	        //Funkcja cykliczna
	        IF NOT #State.inputFlag AND NOT #State.outputFlag THEN
	            IF #Reset THEN
	                #Status.Error := FALSE;
	                #Status.ErrorStatus := 16#0000;
	                IF NOT #Valve.Sensors.In THEN
	                    "changeState"(newState := #S_GO_IN,
	                                  Data := #State);
	                ELSE
	                    "changeState"(newState := #S_IDLE,
	                                  Data := #State);
	                END_IF;
	            END_IF;
	        END_IF;
	        
	        //Funkcja wyjściowa 
	        IF #State.outputFlag THEN
	            ;
	        END_IF;
	        
	    #S_GO_IN:
	        //Funkcja wejścia
	        IF #State.inputFlag AND NOT #State.outputFlag THEN
	            #State.name := 'CHOWANIE SILOWNIKA';
	            #Status.Busy := TRUE;
	            #Status.Ready := FALSE;
	           // #Status.Done := FALSE;
	            #Status.Error := FALSE;
	            #Valve.Coils.In := TRUE;
	            #Valve.Coils.Out := FALSE;
	            RESET_TIMER(#Timers.GoOut.Timer);
	            
	            #Timers.SetIn.IN := TRUE;
	            #Timers.GoOut.IN := TRUE;
	        END_IF;
	        
	        //Funkcja cykliczna
	        IF NOT #State.inputFlag AND NOT #State.outputFlag THEN
	            IF #Valve.Sensors.In AND (NOT #FirstTry OR NOT #SecondPush ) THEN
	                #Execute := FALSE;
	                "changeState"(newState := #S_IDLE,
	                              Data := #State);
	            END_IF;
	            
	            IF #SecondPush AND #FirstTry AND #Timers.GoOut.Timer.Q THEN
	                #FirstTry := FALSE;
	                "changeState"(newState := #S_GO_OUT,
	                              Data := #State);
	            END_IF;
	            
	            
	            
	            IF #Timers.SetIn.Timer.Q THEN
	                #Status.ErrorStatus := #WatchdogIn;
	                "changeState"(newState := #S_ERROR,
	                              Data := #State);
	            END_IF;
	        END_IF;
	        
	        //Funkcja wyjściowa 
	        IF #State.outputFlag THEN
	            #Valve.Coils.In := FALSE;
	            #Timers.SetIn.IN := FALSE;
	            #Timers.GoOut.IN := FALSE;
	        END_IF;
	        
	    #S_GO_OUT:
	        //Funkcja wejścia
	        IF #State.inputFlag AND NOT #State.outputFlag THEN
	            #State.name := 'WYSUNIECIE SILOWNIKA';
	            #Status.Busy := TRUE;
	            #Status.Ready := FALSE;
	            #Status.Done := FALSE;
	            #Status.Error := FALSE;
	            #Valve.Coils.In := FALSE;
	            #Valve.Coils.Out := TRUE;
	            RESET_TIMER(#Timers.Stamping.Timer);
	            RESET_TIMER(#Timers.SetOut.Timer);
	            RESET_TIMER(#Timers.Stamping.Timer);
	            #Timers.SetOut.IN := TRUE;
	        END_IF;
	        
	        //Funkcja cykliczna
	        IF NOT #State.inputFlag AND NOT #State.outputFlag THEN
	            
	            IF #Timers.Stamping.Timer.Q AND #FirstTry THEN
	                #Execute := FALSE;
	                "changeState"(newState := #S_GO_IN,
	                              Data := #State);
	            END_IF;
	            
	            IF #Timers.SecondPush.Timer.Q AND NOT #FirstTry THEN
	                #Execute := FALSE;
	                "changeState"(newState := #S_GO_IN,
	                              Data := #State);
	            END_IF;
	            
	            IF #Timers.SetOut.Timer.Q THEN
	                #Status.ErrorStatus := #WatchdogOut;
	                "changeState"(newState := #S_ERROR,
	                              Data := #State);
	            END_IF;
	        END_IF;
	        
	        //Funkcja wyjściowa 
	        IF #State.outputFlag THEN
	            RESET_TIMER(#Timers.Stamping.Timer);
	            RESET_TIMER(#Timers.SetOut.Timer);
	            RESET_TIMER(#Timers.SecondPush.Timer);
	            #Valve.Coils.Out := FALSE;
	            #Timers.SetOut.IN := FALSE;
	        END_IF;
	END_CASE;
	
	IF (#Timers.SetOut.Timer.ET > #TimerMax AND #FirstTry) THEN
	    #ITV.Sensor.Analog.SetValue := #MaxPreasure;
	ELSIF (#Timers.SetOut.Timer.ET > #TimerSecondPush AND NOT #FirstTry) THEN
	    #ITV.Sensor.Analog.SetValue := #PreasureSecondPush;
	ELSIF #Valve.Coils.In THEN
	    #ITV.Sensor.Analog.SetValue := 3.0;
	ELSE
	    #ITV.Sensor.Analog.SetValue := #RegularPreasure;
	END_IF;
	
	REGION Change state
	    IF #State.inputFlag AND NOT #State.outputFlag THEN
	        #State.inputFlag := FALSE;
	    END_IF;
	    #State.outputFlag := FALSE;
	END_REGION
END_FUNCTION_BLOCK

FUNCTION "changeState" : Void
{ S7_Optimized_Access := 'TRUE' }
VERSION : 0.1
   VAR_INPUT 
      newState : Int;
   END_VAR

   VAR_IN_OUT 
      Data : "s_changeState";
   END_VAR


BEGIN
	IF #Data.state <> #newState THEN
	    #Data.oldState := #Data.state;
	    #Data.state := #newState;
	    #Data.inputFlag := TRUE;
	    #Data.outputFlag := TRUE;
	END_IF;
	
END_FUNCTION

FUNCTION "FC_004_ModularConvoyers" : Void   // FC11, LAD
{ S7_Optimized_Access := 'TRUE' }
// stored: SetENOAutomatically false
BEGIN

REGION Network 1 (SCL)
   //************************************************************
   //===Author: Mateusz Połojko
   //-----Linkedin: https://pl.linkedin.com/in/mateusz-po%C5%82ojko-52a3541b1
   //-----Github: https://github.com/Bhazel95
   //===Description:
   //-----Control of the transporter and executive modules
   //===Customer:
   //-----Apator Powogaz S.A.
   //************************************************************
END_REGION

REGION Network 2
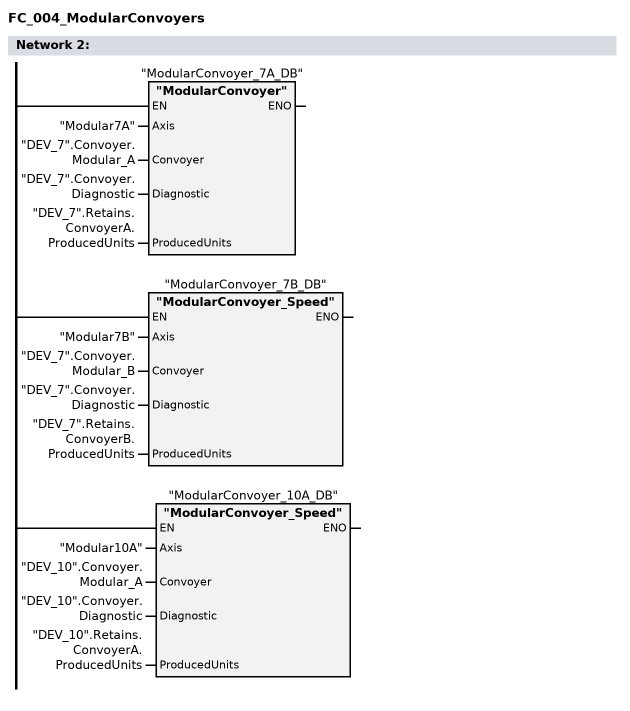
   RUNG wire#powerrail
      "ModularConvoyer_7A_DB"(Axis := "Modular7A", Convoyer := "DEV_7".Convoyer.Modular_A, Diagnostic := "DEV_7".Convoyer.Diagnostic, ProducedUnits := "DEV_7".Retains.ConvoyerA.ProducedUnits)
   END_RUNG
   RUNG wire#powerrail
      "ModularConvoyer_7B_DB"(Axis := "Modular7B", Convoyer := "DEV_7".Convoyer.Modular_B, Diagnostic := "DEV_7".Convoyer.Diagnostic, ProducedUnits := "DEV_7".Retains.ConvoyerB.ProducedUnits)
   END_RUNG
   RUNG wire#powerrail
      "ModularConvoyer_10A_DB"(Axis := "Modular10A", Convoyer := "DEV_10".Convoyer.Modular_A, Diagnostic := "DEV_10".Convoyer.Diagnostic, ProducedUnits := "DEV_10".Retains.ConvoyerA.ProducedUnits)
   END_RUNG
   // the same network as SCL:
   "ModularConvoyer_7A_DB"(Axis := "Modular7A",   // "ModularConvoyer"
                           Convoyer := "DEV_7".Convoyer.Modular_A,
                           Diagnostic := "DEV_7".Convoyer.Diagnostic,
                           ProducedUnits := "DEV_7".Retains.ConvoyerA.ProducedUnits);
   "ModularConvoyer_7B_DB"(Axis := "Modular7B",   // "ModularConvoyer_Speed"
                           Convoyer := "DEV_7".Convoyer.Modular_B,
                           Diagnostic := "DEV_7".Convoyer.Diagnostic,
                           ProducedUnits := "DEV_7".Retains.ConvoyerB.ProducedUnits);
   "ModularConvoyer_10A_DB"(Axis := "Modular10A",   // "ModularConvoyer_Speed"
                           Convoyer := "DEV_10".Convoyer.Modular_A,
                           Diagnostic := "DEV_10".Convoyer.Diagnostic,
                           ProducedUnits := "DEV_10".Retains.ConvoyerA.ProducedUnits);
END_REGION
END_FUNCTION

FUNCTION_BLOCK "ModularConvoyer"
{ S7_Optimized_Access := 'TRUE' }
VERSION : 0.1
   VAR_INPUT 
      Axis {InstructionName := 'TO_PositioningAxis'; LibVersion := '7.0'} : TO_PositioningAxis;
   END_VAR

   VAR_IN_OUT 
      Convoyer : "Modular_10";
      Diagnostic : "DiagnosticMainCabinet";
      ProducedUnits : DInt;
   END_VAR

   VAR 
      R_TRIG_CriticalError {InstructionName := 'R_TRIG'; LibVersion := '1.0'; ExternalAccessible := 'False'; ExternalVisible := 'False'; ExternalWritable := 'False'; S7_SetPoint := 'False'} : R_TRIG;
      R_TRIG_StampingDone {InstructionName := 'R_TRIG'; LibVersion := '1.0'; ExternalAccessible := 'False'; ExternalVisible := 'False'; ExternalWritable := 'False'; S7_SetPoint := 'False'} : R_TRIG;
      R_TRIG_CameraDone {InstructionName := 'R_TRIG'; LibVersion := '1.0'; ExternalAccessible := 'False'; ExternalVisible := 'False'; ExternalWritable := 'False'; S7_SetPoint := 'False'} : R_TRIG;
      R_TRIG_SortingDone {InstructionName := 'R_TRIG'; LibVersion := '1.0'; ExternalAccessible := 'False'; ExternalVisible := 'False'; ExternalWritable := 'False'; S7_SetPoint := 'False'} : R_TRIG;
      R_TRIG_ConvoyerDone {InstructionName := 'R_TRIG'; LibVersion := '1.0'; ExternalAccessible := 'False'; ExternalVisible := 'False'; ExternalWritable := 'False'; S7_SetPoint := 'False'} : R_TRIG;
      R_TRIG_Stop {InstructionName := 'R_TRIG'; LibVersion := '1.0'; ExternalAccessible := 'False'; ExternalVisible := 'False'; ExternalWritable := 'False'; S7_SetPoint := 'False'} : R_TRIG;
      State { S7_SetPoint := 'False'} : "s_changeState";
      Local : Struct
         AutoMode : Bool;
         Buttons : Struct
            START : Bool;
            RESET : Bool;
            STOP : Bool;
         END_STRUCT;
         PermissionToStart : Bool;
         PermissionGoBack : Bool;
         ActionDone : Struct
            Stamping : Bool;
            Camera : Bool;
            Sorting : Bool;
         END_STRUCT;
         Execute : Struct
            Stamping : Bool;
            Camera : Bool;
            Sorting : Bool;
            Convoyer : Bool;
            Blow : Bool;
         END_STRUCT;
         ActionToDo : Struct
            Stamping : Bool;
            Camera : Bool;
            Blow : Bool;
            PreCamera : Array[0..1] of Bool;
         END_STRUCT;
         DoubleStampingDone : Bool;
         StampingTime : Time;
         isMoved : Bool;
         backwardProcess : Bool;
      END_STRUCT;
      Timers : Struct
         WatchdogGoModules { S7_SetPoint := 'False'} : "s_TON";
         WatchdogGoConvoyer : "s_TON";
         Delay : "s_TON";
         DoubleStamp : "s_TON";
         UnloadTimer {InstructionName := 'TON_TIME'; LibVersion := '1.0'; ExternalAccessible := 'False'; ExternalVisible := 'False'; ExternalWritable := 'False'; S7_SetPoint := 'False'} : TON_TIME;
         OskarDelay : "s_TON";
         GoBackwardEnable : "s_TON";
         GoBackward : "s_TON";
      END_STRUCT;
      CameraConnectionTCP_Instance { ExternalAccessible := 'False'; ExternalVisible := 'False'; ExternalWritable := 'False'; S7_SetPoint := 'False'} : "CameraConnectionTCP";
      PositioningAxis_Instance { ExternalAccessible := 'False'; ExternalVisible := 'False'; ExternalWritable := 'False'; S7_SetPoint := 'False'} : "ModularAxis";
      Blow_Instance : "Blow";
      Stamping_Instance : "Stamping";
   END_VAR

   VAR CONSTANT 
      S_IDLE : Int := 0;
      S_ERROR : Int := 20;
      S_GO_CONVOYER : Int := 30;
      S_GO_MODULES : Int := 40;
      S_GO_BACK : Int := 50;
      TEST : Int := 100;
      E_MODULES_TIMEOUT : Word := 16#8000;
      E_CONVOYER_TIMEOUT : Word := 16#8001;
   END_VAR


BEGIN
	//************************************************************
	//===Author: Mateusz Połojko
	//-----Linkedin: https://pl.linkedin.com/in/mateusz-po%C5%82ojko-52a3541b1
	//-----Github: https://github.com/Bhazel95
	//===Description:
	//-----Main function block for convoyer + executive modules control
	//===Customer:
	//-----Apator Powogaz S.A.
	//************************************************************
	
	REGION R/F_TRIG
	    #R_TRIG_CriticalError(CLK := NOT #Convoyer.Safety.SafetyOK OR #PositioningAxis_Instance.Status.Error);
	    #R_TRIG_StampingDone(CLK := #Stamping_Instance.Status.Done);
	    #R_TRIG_CameraDone(CLK := #CameraConnectionTCP_Instance.Status.Done);
	    #R_TRIG_SortingDone(CLK := #Convoyer.SortingStatus.Done);
	    #R_TRIG_ConvoyerDone(CLK := #PositioningAxis_Instance.Status.Ready);
	    #R_TRIG_Stop(CLK := #Local.Buttons.STOP AND #Local.AutoMode);
	END_REGION
	
	REGION Timers
	    //WATCHDOG MACHINE START
	    #Timers.WatchdogGoModules.PT := T#15S;
	    #Timers.WatchdogGoModules.Timer(IN := #Timers.WatchdogGoModules.IN,
	                                    PT := #Timers.WatchdogGoModules.PT);
	    #Timers.WatchdogGoConvoyer.PT := T#10S;
	    #Timers.WatchdogGoConvoyer.Timer(IN := #Timers.WatchdogGoConvoyer.IN,
	                                     PT := #Timers.WatchdogGoConvoyer.PT);
	    #Timers.Delay.PT := T#7S;
	    #Timers.Delay.Timer(IN := #Timers.Delay.IN,
	                        PT := #Timers.Delay.PT);
	    
	    #Timers.DoubleStamp.PT := T#500MS;
	    #Timers.DoubleStamp.Timer(IN := #Timers.DoubleStamp.IN,
	                              PT := #Timers.DoubleStamp.PT);
	    
	    #Timers.OskarDelay.PT := T#5000MS;
	    #Timers.OskarDelay.Timer(IN := #Timers.OskarDelay.IN,
	                             PT := #Timers.OskarDelay.PT);
	    
	    #Timers.GoBackwardEnable.PT := T#3000MS;
	    #Timers.GoBackwardEnable.Timer(IN := #Convoyer.ButtonControl.ButtonBoxLeft.ButtonReset OR #Convoyer.ButtonControl.ButtonBoxRight.ButtonReset,
	                                   PT := #Timers.GoBackwardEnable.PT);
	    
	    #Timers.GoBackward.PT := T#2000MS;
	    #Timers.GoBackward.Timer(IN := #Timers.GoBackward.IN,
	                             PT := #Timers.GoBackward.PT);
	    
	    #Timers.UnloadTimer(IN := NOT #Convoyer.Sensors.UnloadingPresence,
	                        PT := T#1000MS);
	END_REGION
	
	//Permission to start
	#Local.PermissionToStart := #Diagnostic.DiagnosticOK AND NOT #Convoyer.Alarms.Fault24V AND #Convoyer.Safety.SafetyOK
	AND NOT #Convoyer.Alarms.Present AND #Convoyer.Pneumatics.Stamping.Sensors.In AND #Convoyer.Safety.LightCurtain_Stamping
	AND NOT #Convoyer.Pneumatics.Stamping.Sensors.Out AND (#Convoyer.CameraStatus.Ready OR NOT #Convoyer.HMI.Camera.Enable)
	AND #Convoyer.MotorStatus.Ready AND #Convoyer.Sensors.Stamp_Check_1 AND #Convoyer.Sensors.UnloadingPresence AND #Convoyer.Sensors.Span;
	
	#Local.PermissionGoBack := #Diagnostic.DiagnosticOK AND #Convoyer.Safety.SafetyOK
	AND NOT #Convoyer.Alarms.Present AND #Convoyer.Pneumatics.Stamping.Sensors.In
	AND NOT #Convoyer.Pneumatics.Stamping.Sensors.Out AND #Convoyer.MotorStatus.Ready AND #Convoyer.Sensors.Stamp_Check_1 AND #Convoyer.Sensors.UnloadingPresence AND #Convoyer.Sensors.Span AND #Convoyer.Sensors.JogBack;
	
	//Start button
	#Local.Buttons.START := #Convoyer.ButtonControl.ButtonBoxLeft.ButtonStart OR #Convoyer.ButtonControl.ButtonBoxRight.ButtonStart OR #Convoyer.HMI.Buttons.Start;
	//Stop button
	#Local.Buttons.STOP := #Convoyer.ButtonControl.ButtonBoxLeft.ButtonStop OR #Convoyer.ButtonControl.ButtonBoxRight.ButtonStop OR #Convoyer.HMI.Buttons.Stop;
	//Reset button
	#Local.Buttons.RESET := #Convoyer.ButtonControl.ButtonBoxLeft.ButtonReset OR #Convoyer.ButtonControl.ButtonBoxRight.ButtonReset OR #Convoyer.ButtonControl.CabinetBox.ButtonReset;
	
	CASE #State.state OF
	    #S_IDLE:
	        //Funkcja wejścia
	        IF #State.inputFlag AND NOT #State.outputFlag THEN
	            #Convoyer.ConvoyerStatus.Busy := FALSE;
	            #Convoyer.ConvoyerStatus.Done := FALSE;
	            #Convoyer.ConvoyerStatus.Error := FALSE;
	            #Convoyer.ConvoyerStatus.ErrorStatus := 16#0000;
	            #Convoyer.ConvoyerStatus.Ready := TRUE;
	        END_IF;
	        
	        //Funkcja cykliczna
	        IF NOT #State.inputFlag AND NOT #State.outputFlag THEN
	            //ZABEZPIECZENIE PRZED MANUALNYM RUSZENIEM TRANSPORTERA
	            IF #Convoyer.MotorControl.MC_MOVEJOG.JogBackward OR #Convoyer.MotorControl.MC_MOVEJOG.JogForward THEN
	                #Local.isMoved := TRUE;
	            END_IF;
	            IF #Convoyer.Safety.LightCurtain_Stamping AND #Local.PermissionToStart AND (#Local.Buttons.START OR #Local.AutoMode) AND NOT #Local.Buttons.STOP AND NOT #Local.Buttons.RESET THEN
	                #Local.AutoMode := TRUE;
	                IF ((NOT #Convoyer.Sensors.StampingPresence AND NOT #Local.ActionDone.Stamping) OR (NOT #Convoyer.Sensors.CameraPresence AND NOT #Local.ActionDone.Camera)) AND NOT #Local.isMoved THEN
	                    "changeState"(newState := #S_GO_MODULES,
	                                  Data := #State);
	                ELSIF ((#Local.ActionDone.Stamping OR #Convoyer.Sensors.StampingPresence) AND (#Local.ActionDone.Camera OR #Convoyer.Sensors.CameraPresence)) OR #Local.isMoved THEN
	                    "changeState"(newState := #S_GO_CONVOYER,
	                                  Data := #State);
	                END_IF;
	            END_IF;
	            //COFANIE TRANSPORTERA
	            IF NOT #Local.AutoMode AND #Local.PermissionGoBack AND #Timers.GoBackwardEnable.Timer.Q AND NOT #Local.Buttons.START AND NOT #Local.Buttons.STOP THEN
	                #Local.isMoved := TRUE;
	                "changeState"(newState := #S_GO_BACK,
	                              Data := #State);
	            END_IF;
	            
	        END_IF;
	        
	        //Funkcja wyjściowa 
	        IF #State.outputFlag THEN
	            #Convoyer.ConvoyerStatus.Ready := FALSE;
	            #Convoyer.ConvoyerStatus.Busy := TRUE;
	        END_IF;
	        
	    #S_ERROR:
	        //Funkcja wejścia
	        IF #State.inputFlag AND NOT #State.outputFlag THEN
	            #Convoyer.ConvoyerStatus.Busy := FALSE;
	            #Convoyer.ConvoyerStatus.Done := FALSE;
	            #Convoyer.ConvoyerStatus.Error := TRUE;
	            #Convoyer.ConvoyerStatus.Ready := FALSE;
	            #Timers.WatchdogGoConvoyer.IN := FALSE;
	            #Timers.WatchdogGoModules.IN := FALSE;
	            #Local.Execute.Convoyer := FALSE;
	            #Local.Execute.Stamping := FALSE;
	            #Local.Execute.Camera := FALSE;
	            //#Local.ActionDone.Camera := FALSE;
	            #Local.AutoMode := FALSE;
	        END_IF;
	        
	        //Funkcja cykliczna
	        IF NOT #State.inputFlag AND NOT #State.outputFlag THEN
	            IF #Local.Buttons.RESET AND NOT #Convoyer.Alarms.Present AND #Convoyer.Safety.SafetyOK
	                AND (#CameraConnectionTCP_Instance.Status.Ready OR NOT #Convoyer.HMI.Camera.Enable) AND #PositioningAxis_Instance.Status.Ready
	                AND (#Stamping_Instance.Status.Ready OR NOT #Convoyer.HMI.Stamping.Enable) AND #Local.PermissionToStart THEN
	                #Convoyer.ConvoyerStatus.Error := FALSE;
	                "changeState"(newState := #S_IDLE,
	                              Data := #State);
	            END_IF;
	        END_IF;
	        
	        //Funkcja wyjściowa 
	        IF #State.outputFlag THEN
	            ;
	        END_IF;
	        
	    #S_GO_CONVOYER:
	        //Funkcja wejścia
	        IF #State.inputFlag AND NOT #State.outputFlag THEN
	            #Timers.WatchdogGoConvoyer.IN := TRUE;
	            #Local.ActionDone.Stamping := FALSE;
	            #Local.ActionDone.Camera := FALSE;
	            #Local.ActionDone.Sorting := FALSE;
	            #Local.ActionToDo.PreCamera[1] := #Local.ActionToDo.PreCamera[0];
	            #Local.Execute.Convoyer := TRUE;
	        END_IF;
	        
	        //Funkcja cykliczna
	        IF NOT #State.inputFlag AND NOT #State.outputFlag THEN
	            IF #R_TRIG_ConvoyerDone.Q THEN
	                #Local.isMoved := FALSE;
	                IF NOT #Local.AutoMode OR NOT #Convoyer.Safety.LightCurtain_Stamping THEN
	                    "changeState"(newState := #S_IDLE,
	                                  Data := #State);
	                ELSE
	                    "changeState"(newState := #S_GO_MODULES,
	                                  Data := #State);
	                END_IF;
	            END_IF;
	            IF #PositioningAxis_Instance.Status.Error THEN
	                "changeState"(newState := #S_ERROR,
	                              Data := #State);
	            END_IF;
	            //WATCHDOG
	            IF #Timers.WatchdogGoConvoyer.Timer.Q THEN
	                #PositioningAxis_Instance.Status.ErrorStatus := #E_CONVOYER_TIMEOUT;
	                "changeState"(newState := #S_ERROR,
	                              Data := #State);
	            END_IF;
	        END_IF;
	        
	        //Funkcja wyjściowa 
	        IF #State.outputFlag THEN
	            #Local.Execute.Convoyer := FALSE;
	            #Local.ActionDone.Stamping := FALSE;
	            #Local.ActionDone.Camera := FALSE;
	            #Local.ActionDone.Sorting := FALSE;
	            #Timers.WatchdogGoConvoyer.IN := FALSE;
	            #Local.Execute.Convoyer := FALSE;
	        END_IF;
	        
	    #S_GO_MODULES:
	        //Funkcja wejścia
	        IF #State.inputFlag AND NOT #State.outputFlag THEN
	            #Timers.OskarDelay.IN := TRUE;
	            #Timers.WatchdogGoModules.IN := TRUE;
	            #Timers.Delay.IN := TRUE;
	            #Local.DoubleStampingDone := FALSE;
	            IF #Convoyer.HMI.Stamping.Double THEN
	                #Local.StampingTime := T#1MS;
	            ELSE
	                #Local.StampingTime := #Convoyer.HMI.Stamping.TimerStamping;
	            END_IF;
	            #Local.Execute.Blow := #Convoyer.Sensors.BlowPresence AND #Convoyer.HMI.Blow.Enable;
	            #Local.Execute.Stamping := NOT #Local.ActionDone.Stamping AND NOT #Convoyer.Sensors.StampingPresence AND #Convoyer.HMI.Stamping.Enable;
	            
	            //TUTAJ NA DOLE
	            #Local.Execute.Camera := ((NOT #Local.ActionDone.Camera AND NOT #Convoyer.Sensors.CameraPresence) OR (#Local.ActionToDo.PreCamera[1] AND NOT #Local.ActionDone.Camera)) AND #Convoyer.HMI.Camera.Enable;
	            #Local.ActionToDo.Stamping := #Local.Execute.Stamping;
	            #Local.ActionToDo.Camera := #Local.Execute.Camera;
	            #Local.ActionToDo.PreCamera[0] := #Convoyer.Sensors.BlowPresence; //DODANE ABY ZOBACZYC CZY WYELIMINUJE BLAD BRAKU ZDJEC
	        END_IF;
	        //Funkcja cykliczna
	        IF NOT #State.inputFlag AND NOT #State.outputFlag THEN
	            REGION double stamping
	                IF #Convoyer.HMI.Stamping.Double AND NOT #Local.DoubleStampingDone AND #Timers.DoubleStamp.Timer.Q THEN
	                    #Local.StampingTime := #Convoyer.HMI.Stamping.TimerStamping;
	                    #Local.DoubleStampingDone := TRUE;
	                    #Local.Execute.Stamping := TRUE;
	                END_IF;
	            END_REGION
	            
	            IF #R_TRIG_CameraDone.Q THEN
	                #Local.ActionDone.Camera := TRUE;
	                #Local.ActionToDo.Camera := FALSE;
	                #Local.Execute.Camera := FALSE;
	            END_IF;
	            IF #R_TRIG_SortingDone.Q THEN
	                #Local.ActionDone.Sorting := TRUE;
	            END_IF;
	            IF #R_TRIG_StampingDone.Q THEN
	                #ProducedUnits := #ProducedUnits + 1;
	                IF NOT #Convoyer.HMI.Stamping.Double THEN
	                    #Local.ActionDone.Stamping := TRUE;
	                    #Local.ActionToDo.Stamping := FALSE;
	                    #Local.Execute.Stamping := FALSE;
	                ELSIF #Convoyer.HMI.Stamping.Double AND NOT #Local.DoubleStampingDone THEN
	                    #Timers.DoubleStamp.IN := TRUE;
	                    #Local.Execute.Stamping := FALSE;
	                ELSIF #Convoyer.HMI.Stamping.Double AND #Local.DoubleStampingDone THEN
	                    #Local.ActionDone.Stamping := TRUE;
	                    #Local.ActionToDo.Stamping := FALSE;
	                    #Local.Execute.Stamping := FALSE;
	                END_IF;
	            END_IF;
	            
	            //Oczekiwanie na potwierdzenia blokow  - komentarz -->> opoznienie zalaczenia ruchu stolu dla Oskara
	            IF (#Local.ActionDone.Stamping OR NOT #Local.ActionToDo.Stamping) AND (#Local.ActionDone.Camera OR NOT #Local.ActionToDo.Camera) AND NOT #Local.Execute.Blow (* AND #Timers.OskarDelay.Timer.Q *)THEN
	                IF NOT #Local.AutoMode THEN
	                    "changeState"(newState := #S_IDLE,
	                                  Data := #State);
	                ELSE
	                    IF #Local.PermissionToStart THEN
	                        "changeState"(newState := #S_GO_CONVOYER,
	                                      Data := #State);
	                    ELSE
	                        "changeState"(newState := #S_IDLE,
	                                      Data := #State);
	                    END_IF;
	                END_IF;
	            END_IF;
	            //Modules Error
	            IF (#CameraConnectionTCP_Instance.Status.Error OR #Stamping_Instance.Status.Error) AND #Timers.Delay.Timer.Q THEN
	                "changeState"(newState := #S_ERROR,
	                              Data := #State);
	            END_IF;
	            
	            //WATCHDOG
	            IF #Timers.WatchdogGoModules.Timer.Q THEN
	                #PositioningAxis_Instance.Status.ErrorStatus := #E_MODULES_TIMEOUT;
	                "changeState"(newState := #S_ERROR,
	                              Data := #State);
	            END_IF;
	        END_IF;
	        
	        //Funkcja wyjściowa 
	        IF #State.outputFlag THEN
	            #Timers.Delay.IN := FALSE;
	            #Timers.OskarDelay.IN := FALSE;
	            #Timers.DoubleStamp.IN := FALSE;
	            #Timers.WatchdogGoModules.IN := FALSE;
	            #Local.Execute.Stamping := FALSE;
	            #Local.Execute.Camera := FALSE;
	            #Local.Execute.Sorting := FALSE;
	        END_IF;
	        
	    #S_GO_BACK:
	        //Funkcja wejścia
	        IF #State.inputFlag AND NOT #State.outputFlag THEN
	            #Local.backwardProcess := TRUE;
	            #Timers.GoBackward.IN := TRUE;
	            #Local.isMoved := TRUE;
	            #Convoyer.MotorControl.MC_MOVEJOG.JogBackward := TRUE;
	            
	        END_IF;
	        
	        //Funkcja cykliczna
	        IF NOT #State.inputFlag AND NOT #State.outputFlag THEN
	            IF (#Timers.GoBackward.Timer.Q AND #Convoyer.Safety.LightCurtain_Stamping) OR NOT #Convoyer.Sensors.JogBack THEN
	                #Convoyer.MotorControl.MC_MOVEJOG.JogBackward := FALSE;
	                "changeState"(newState := #S_IDLE,
	                              Data := #State);
	            END_IF;
	        END_IF;
	        
	        //Funkcja wyjściowa 
	        IF #State.outputFlag THEN
	            #Local.backwardProcess := FALSE;
	            #Convoyer.MotorControl.MC_MOVEJOG.JogBackward := FALSE;
	            #Timers.GoBackward.IN := FALSE;
	        END_IF;
	        
	END_CASE;
	
	REGION FunctionBlocks
	    #Stamping_Instance(Reset := #Local.Buttons.RESET,
	                       SecondPush := #Convoyer.HMI.Stamping.SecondPush,
	                       TimerSecondPush := #Convoyer.HMI.Stamping.TimerSecond,
	                       PreasureSecondPush := #Convoyer.HMI.Stamping.SecondPreasure,
	                       TimerStamp := #Convoyer.HMI.Stamping.TimerStamping,
	                       TimerMax := #Convoyer.HMI.Stamping.TimerMaxPreasure,
	                       MaxPreasure := #Convoyer.HMI.Stamping.MaxPreasure,
	                       RegularPreasure := #Convoyer.HMI.Stamping.RegularPreasure,
	                       Status => #Convoyer.StampingStatus,
	                       Valve := #Convoyer.Pneumatics.Stamping,
	                       ITV := #Convoyer.Pneumatics.IVT,
	                       Execute := #Local.Execute.Stamping);
	    #CameraConnectionTCP_Instance(Enable := #Convoyer.HMI.Camera.Enable,
	                                  Execute := #Local.Execute.Camera,
	                                  Reset := #Local.Buttons.RESET,
	                                  ConnectionTimer := #Convoyer.HMI.Camera.TimerConnection,
	                                  Status => #Convoyer.CameraStatus,
	                                  Parameters := #Convoyer.CameraConnection);
	    #PositioningAxis_Instance(HomingSensor := #Convoyer.Sensors.Homing_I,
	                              Reset := #Local.Buttons.RESET,
	                              InverterOK := #Convoyer.Safety.InverterOK,
	                              Axis := #Axis,
	                              Status => #Convoyer.MotorStatus,
	                              Execute := #Local.Execute.Convoyer,
	                              PositioningAxis := #Convoyer.MotorControl);
	    #Blow_Instance(Timer := #Convoyer.HMI.Blow."Time",
	                   Execute := #Local.Execute.Blow,
	                   Coil := #Convoyer.Pneumatics.Valve.Coils.Out);
	END_REGION
	
	REGION Lights
	    //RESET BUTTON
	    #Convoyer.ButtonControl.ButtonBoxLeft.LightReset := #Convoyer.ConvoyerStatus.Error OR #Convoyer.CameraStatus.Error OR #Convoyer.StampingStatus.Error OR #Convoyer.MotorStatus.Error OR (NOT #Convoyer.Pneumatics.Stamping.Sensors.In AND #Convoyer.StampingStatus.Ready) OR (#Local.backwardProcess AND "Clock_1Hz");
	    #Convoyer.ButtonControl.ButtonBoxRight.LightReset := #Convoyer.ConvoyerStatus.Error OR #Convoyer.CameraStatus.Error OR #Convoyer.StampingStatus.Error OR #Convoyer.MotorStatus.Error OR (NOT #Convoyer.Pneumatics.Stamping.Sensors.In AND #Convoyer.StampingStatus.Ready) OR (#Local.backwardProcess AND "Clock_1Hz");
	    #Convoyer.ButtonControl.CabinetBox.LightReset := #Convoyer.ConvoyerStatus.Error OR #Convoyer.CameraStatus.Error OR #Convoyer.StampingStatus.Error OR #Convoyer.MotorStatus.Error OR (NOT #Convoyer.Pneumatics.Stamping.Sensors.In AND #Convoyer.StampingStatus.Ready);
	    //STOP BUTTON
	    #Convoyer.ButtonControl.ButtonBoxLeft.LightStop := #Convoyer.ConvoyerStatus.Busy AND NOT #Local.AutoMode;
	    #Convoyer.ButtonControl.ButtonBoxRight.LightStop := #Convoyer.ConvoyerStatus.Busy AND NOT #Local.AutoMode;
	    //START BUTTON
	    #Convoyer.ButtonControl.ButtonBoxLeft.LightStart := #Convoyer.ConvoyerStatus.Ready AND #Local.PermissionToStart AND NOT #Local.AutoMode;
	    #Convoyer.ButtonControl.ButtonBoxRight.LightStart := #Convoyer.ConvoyerStatus.Ready AND #Local.PermissionToStart AND NOT #Local.AutoMode;
	    //ANDON 
	    #Convoyer.Lights.Red := #Convoyer.ConvoyerStatus.Error OR #Convoyer.CameraStatus.Error OR #Convoyer.StampingStatus.Error OR #Convoyer.MotorStatus.Error;
	    #Convoyer.Lights.Green := #Convoyer.ConvoyerStatus.Busy OR #Local.AutoMode;
	    #Convoyer.Lights.Blue := #Convoyer.ConvoyerStatus.Ready AND #Local.PermissionToStart AND NOT #Local.AutoMode;
	    #Convoyer.Lights.Orange := #Timers.UnloadTimer.Q;
	END_REGION
	
	//Set AutoMode off
	IF #R_TRIG_Stop.Q THEN
	    #Local.AutoMode := FALSE;
	END_IF;
	
	//Error trig
	IF #R_TRIG_CriticalError.Q THEN
	    IF NOT #PositioningAxis_Instance.Status.Done THEN
	        #Local.isMoved := TRUE;
	    END_IF;
	    
	    "changeState"(newState := #S_ERROR,
	                  Data := #State);
	END_IF;
	
	REGION Change state
	    IF #State.inputFlag AND NOT #State.outputFlag THEN
	        #State.inputFlag := FALSE;
	    END_IF;
	    #State.outputFlag := FALSE;
	END_REGION
END_FUNCTION_BLOCK

FUNCTION_BLOCK "CameraConnectionTCP"   // FB2, LAD
{ S7_Optimized_Access := 'TRUE' }
// stored: MemoryReserve 100, SetENOAutomatically false
   VAR_INPUT
      Enable : Bool;
      Execute : Bool;
      Reset : Bool;
      ConnectionTimer : Time;
   END_VAR
   VAR_OUTPUT
      Status : "Status";
   END_VAR
   VAR_IN_OUT
      Parameters : TCON_IP_v4;
   END_VAR
   VAR
      TCON_Instance { ExternalAccessible := 'False'; ExternalVisible := 'False'; ExternalWritable := 'False'} : TCON;
      TDISCON_Instance { ExternalAccessible := 'False'; ExternalVisible := 'False'; ExternalWritable := 'False'} : TDISCON;
      TRCV_Instance { ExternalAccessible := 'False'; ExternalVisible := 'False'; ExternalWritable := 'False'} : TRCV;
      TSEND_Instance { ExternalAccessible := 'False'; ExternalVisible := 'False'; ExternalWritable := 'False'} : TSEND;
      Connection : Struct
         TCON : Struct
            REQ : Bool;
            BUSY : Bool;
            DONE : Bool;
            ERROR : Bool;
            STATUS : Word;
            CONNECTION_DATA : Struct
               InterfaceID : HW_ANY := 64;
               ID : HW_ANY := 1;
               ConnectionType : Byte := 16#0B;
               ActiveEstablished : Bool := false;
               RemodeAddress { S7_SetPoint := 'True'} : IP_V4;
               RemotePort : UInt;
               LocalPort : UInt := 2000;
            END_STRUCT;
         END_STRUCT;
         TDISCON : Struct
            REQ : Bool;
            BUSY : Bool;
            DONE : Bool;
            ERROR : Bool;
            STATUS : Word;
         END_STRUCT;
         TSEND : Struct
            REQ : Bool;
            LEN : UDInt;
            BUSY : Bool;
            DONE : Bool;
            ERROR : Bool;
            STATUS : Word;
         END_STRUCT;
         TRVC : Struct
            ENABLE : Bool;
            ADHOC : Bool := TRUE;
            LEN : UDInt;
            NDR : Bool;
            BUSY : Bool;
            RVC_LEN : UDInt;
            ERROR : Bool;
            STATUS : Word;
         END_STRUCT;
      END_STRUCT;
      Data : Struct
         RVC : Array[0..999] of Byte;
         SEND : Array[0..999] of Byte;
      END_STRUCT;
      State : "s_changeState";
      Timers : Struct
         WatchdogInit : "s_TON";
         WatchdogCamera : "s_TON";
         WatchdogInitRVC { S7_SetPoint := 'True'} : "s_TON";
         WatchdogMachineStart { S7_SetPoint := 'True'} : "s_TON";
      END_STRUCT;
      MessageGenerating : Struct
         i : Int;
         len : DInt;
         "string" : String[100];
         chars : Array[0..99] of Char;
      END_STRUCT;
      Local : Struct
         MessageSent : Bool;
         MessageSentCounter : SInt;
         prevState : Int;
      END_STRUCT;
      F_TRIG_Enable { ExternalAccessible := 'False'; ExternalVisible := 'False'; ExternalWritable := 'False'} : F_TRIG;
      R_TRIG_Execute { ExternalAccessible := 'False'; ExternalVisible := 'False'; ExternalWritable := 'False'} : R_TRIG;
      R_TRIG_Enable { ExternalAccessible := 'False'; ExternalVisible := 'False'; ExternalWritable := 'False'} : R_TRIG;
      Connected : Bool;
      DebugCounter : DInt;
   END_VAR
   VAR CONSTANT
      S_INITIALIZE : Int := 1;
      S_DISCONNECT : Int := 10;
      S_ERROR : Int := 20;
      S_ENABLE_RVC : Int := 30;
      S_MACHINE_START : Int := 40;
      S_IDLE : Int := 50;
      S_START_CAMERA : Int := 60;
      S_REPEAT : Int := 70;
      STATE_TEST : Int := 100;
      COMAND_SEND_MACHINE_START : String := 'command: machine_start';
      COMMAND_RVC_MACHINE_START : String := 'command: camera_ready';
      COMMAND_SEND_START_CONTROL : String := 'command: start_control';
      COMMAND_RVC_CONTROL_DONE : String := 'command: control_done';
      E_CONNECTION_TIMEOUT : Word := 16#8000;
      E_WRONG_RESPONSE_MACHINE_START : Word := 16#8001;
      E_START_MACHINE_NOT_SENT : Word := 16#8002;
      E_START_MACHINE_NO_RESPONSE : Word := 16#8003;
      E_WRONG_RESPONSE_CAMERA : Word := 16#8004;
      E_CAMERA_NO_RESPONSE : Word := 16#8005;
      E_CAMERA_NOT_SENT : Word := 16#8006;
      E_TRCV_ERROR : Word := 16#8007;
      E_TRCV_TIMEOUT : Word := 16#8008;
      E_TCON_ERROR : Word := 16#8009;
      E_TDISCON_ERROR : Word := 16#8010;
      E_TSEND_ERROR : Word := 16#8011;
   END_VAR
   // Connection.TCON.CONNECTION_DATA.RemodeAddress.ADDR[1] := 192;
   // Connection.TCON.CONNECTION_DATA.RemodeAddress.ADDR[2] := 168;
   // Connection.TCON.CONNECTION_DATA.RemodeAddress.ADDR[3] := 0;
   // Connection.TCON.CONNECTION_DATA.RemodeAddress.ADDR[4] := 69;
BEGIN

REGION Network 1 (SCL)
   //************************************************************
   //===Author: Mateusz Połojko
   //-----Linkedin: https://pl.linkedin.com/in/mateusz-po%C5%82ojko-52a3541b1
   //-----Github: https://github.com/Bhazel95
   //===Description:
   //-----Camera control via TCP/IP
   //===Customer:
   //-----Apator Powogaz S.A.
   //************************************************************
END_REGION

REGION Network 2
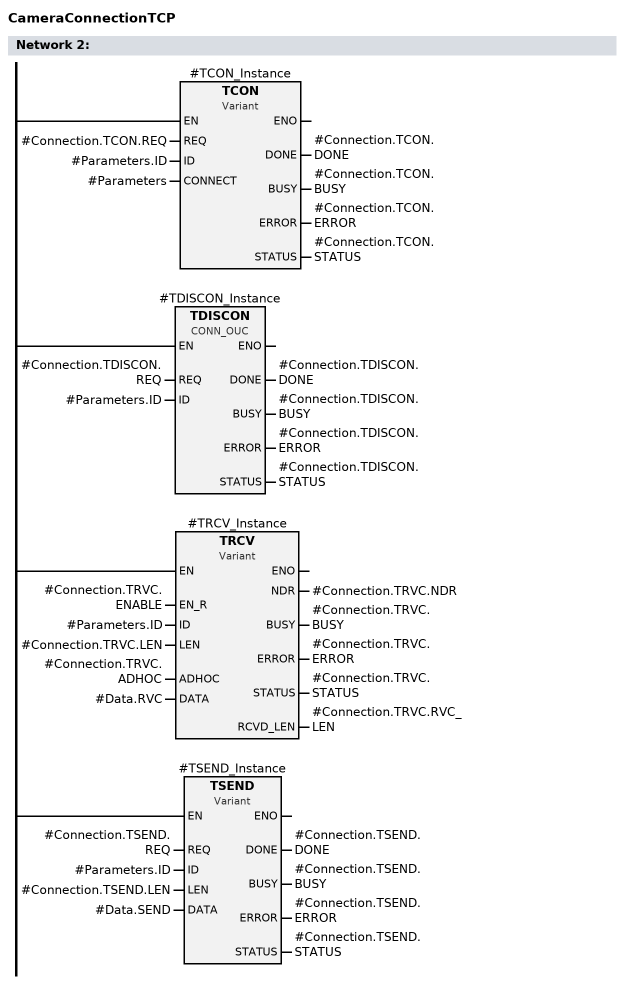
   RUNG wire#powerrail
      { S7_Templates := "[con_type := Variant, id_type := CONN_OUC]" } #TCON_Instance.TCON(REQ := #Connection.TCON.REQ, ID := #Parameters.ID, CONNECT := #Parameters, DONE => #Connection.TCON.DONE, BUSY => #Connection.TCON.BUSY, ERROR => #Connection.TCON.ERROR, STATUS => #Connection.TCON.STATUS)
   END_RUNG
   RUNG wire#powerrail
      { S7_Templates := "id_type := CONN_OUC" } #TDISCON_Instance.TDISCON(REQ := #Connection.TDISCON.REQ, ID := #Parameters.ID, DONE => #Connection.TDISCON.DONE, BUSY => #Connection.TDISCON.BUSY, ERROR => #Connection.TDISCON.ERROR, STATUS => #Connection.TDISCON.STATUS)
   END_RUNG
   RUNG wire#powerrail
      { S7_Templates := "[card := 1, ptr_type := Variant, value_type := UDInt, id_type := CONN_OUC]" } #TRCV_Instance.TRCV(EN_R := #Connection.TRVC.ENABLE, ID := #Parameters.ID, LEN := #Connection.TRVC.LEN, ADHOC := #Connection.TRVC.ADHOC, DATA := #Data.RVC, NDR => #Connection.TRVC.NDR, BUSY => #Connection.TRVC.BUSY, ERROR => #Connection.TRVC.ERROR, STATUS => #Connection.TRVC.STATUS, RCVD_LEN => #Connection.TRVC.RVC_LEN)
   END_RUNG
   RUNG wire#powerrail
      { S7_Templates := "[data_type := Variant, len_type := UDInt, id_type := CONN_OUC]" } #TSEND_Instance.TSEND(REQ := #Connection.TSEND.REQ, ID := #Parameters.ID, LEN := #Connection.TSEND.LEN, DATA := #Data.SEND, DONE => #Connection.TSEND.DONE, BUSY => #Connection.TSEND.BUSY, ERROR => #Connection.TSEND.ERROR, STATUS => #Connection.TSEND.STATUS)
   END_RUNG
   // the same network as SCL:
   #TCON_Instance(REQ := #Connection.TCON.REQ,   // TCON
                  ID := #Parameters.ID,
                  CONNECT := #Parameters,
                  DONE => #Connection.TCON.DONE,
                  BUSY => #Connection.TCON.BUSY,
                  ERROR => #Connection.TCON.ERROR,
                  STATUS => #Connection.TCON.STATUS);
   #TDISCON_Instance(REQ := #Connection.TDISCON.REQ,   // TDISCON
                     ID := #Parameters.ID,
                     DONE => #Connection.TDISCON.DONE,
                     BUSY => #Connection.TDISCON.BUSY,
                     ERROR => #Connection.TDISCON.ERROR,
                     STATUS => #Connection.TDISCON.STATUS);
   #TRCV_Instance(EN_R := #Connection.TRVC.ENABLE,   // TRCV
                  ID := #Parameters.ID,
                  LEN := #Connection.TRVC.LEN,
                  ADHOC := #Connection.TRVC.ADHOC,
                  DATA := #Data.RVC,
                  NDR => #Connection.TRVC.NDR,
                  BUSY => #Connection.TRVC.BUSY,
                  ERROR => #Connection.TRVC.ERROR,
                  STATUS => #Connection.TRVC.STATUS,
                  RCVD_LEN => #Connection.TRVC.RVC_LEN);
   #TSEND_Instance(REQ := #Connection.TSEND.REQ,   // TSEND
                   ID := #Parameters.ID,
                   LEN := #Connection.TSEND.LEN,
                   DATA := #Data.SEND,
                   DONE => #Connection.TSEND.DONE,
                   BUSY => #Connection.TSEND.BUSY,
                   ERROR => #Connection.TSEND.ERROR,
                   STATUS => #Connection.TSEND.STATUS);
END_REGION

REGION Network 3 (SCL)
   REGION TIMERS
       //WATCHDOG INICJALIZACJA POŁĄCZENIA
       #Timers.WatchdogInit.PT := #ConnectionTimer;
       #Timers.WatchdogInit.Timer(IN := #Timers.WatchdogInit.IN,
                                  PT := #Timers.WatchdogInit.PT);

       //WATCHDOG WYSYLANIE DANYCH DO ZROBIENIA ZDJĘCIA
       #Timers.WatchdogCamera.PT := T#5S;
       #Timers.WatchdogCamera.Timer(IN := #Timers.WatchdogCamera.IN,
                                    PT := #Timers.WatchdogCamera.PT);

       //WATCHDOG INICJALIZACJI POŁĄCZENIA
       #Timers.WatchdogInitRVC.PT := T#10S;
       #Timers.WatchdogInitRVC.Timer(IN := #Timers.WatchdogInitRVC.IN,
                                     PT := #Timers.WatchdogInitRVC.PT);

       //WATCHDOG MACHINE START
       #Timers.WatchdogMachineStart.PT := T#10S;
       #Timers.WatchdogMachineStart.Timer(IN := #Timers.WatchdogMachineStart.IN,
                                          PT := #Timers.WatchdogMachineStart.PT);
   END_REGION

   REGION R/F TRIG
       #F_TRIG_Enable(CLK:=#Enable);
       #R_TRIG_Execute(CLK:=#Execute);
       #R_TRIG_Enable(CLK:=#Enable);
   END_REGION


   CASE #State.state OF
       #S_INITIALIZE:
           //Funkcja wejścia
           IF #State.inputFlag AND NOT #State.outputFlag THEN
               #State.name := 'INICJALIZACJA POLACZENIA';
              // #State.name := 'ERROR';
               #Status.Busy := TRUE;
               #Status.Ready := FALSE;
               #Status.Done := FALSE;
               #Status.Error := FALSE;
               #Status.ErrorStatus := 16#0000;
               #Timers.WatchdogCamera.IN := FALSE;
               #Timers.WatchdogInit.IN := FALSE;
               #Timers.WatchdogInitRVC.IN := FALSE;
               #Timers.WatchdogMachineStart.IN := FALSE;
               #Connection.TRVC.ADHOC := TRUE;
               #Connection.TCON.REQ := TRUE;
               #Timers.WatchdogInit.IN := TRUE;
               #Connection.TCON.REQ := TRUE;
           END_IF;

           //Funkcja cykliczna
           IF NOT #State.inputFlag AND NOT #State.outputFlag THEN
               IF #Connection.TCON.STATUS = 16#0000 (* AND NOT #Connection.TCON.BUSY *) THEN
                   "changeState"(newState := #S_ENABLE_RVC,
                                 Data := #State);
               END_IF;

               IF #Timers.WatchdogInit.Timer.Q THEN
                   #Status.ErrorStatus  := #E_CONNECTION_TIMEOUT;
                   "changeState"(newState := #S_ERROR,
                                 Data := #State);
               END_IF;
           END_IF;

           //Funkcja wyjściowa 
           IF #State.outputFlag THEN
               #Timers.WatchdogInit.IN := FALSE;
           END_IF;

       #S_DISCONNECT:
           //Funkcja wejścia
           IF #State.inputFlag AND NOT #State.outputFlag THEN
               #State.name := 'DISCONNECT Z SIECIA';
               #Status.ErrorStatus  := 16#0000;
               #Connection.TCON.REQ := FALSE;
               #Connection.TSEND.REQ := FALSE;
               #Connection.TRVC.ENABLE := FALSE;
               #Connection.TDISCON.REQ := TRUE;
               #Status.ErrorStatus := 16#0000;
               #Timers.WatchdogCamera.IN := FALSE;
               #Timers.WatchdogInit.IN := FALSE;
               #Timers.WatchdogInitRVC.IN := FALSE;
               #Timers.WatchdogMachineStart.IN := FALSE;
               #Status.Error := FALSE;
           END_IF;

           //Funkcja cykliczna
           IF NOT #State.inputFlag AND NOT #State.outputFlag THEN
               IF NOT #Connection.TDISCON.BUSY AND NOT #Connection.TCON.BUSY THEN
                   #Connection.TDISCON.REQ := FALSE;
               END_IF;
               IF #Enable AND #Connection.TDISCON.REQ = FALSE  THEN
                   "changeState"(newState := #S_INITIALIZE,
                                 Data := #State);
               END_IF;
           END_IF;

           //Funkcja wyjściowa 
           IF #State.outputFlag THEN
               ;
           END_IF;

       #S_ERROR:
           //Funkcja wejścia
           IF #State.inputFlag AND NOT #State.outputFlag THEN
               #State.name := 'ERROR';
               #Status.Busy := FALSE;
               #Status.Ready := FALSE;
               #Status.Done := FALSE;
               #Status.Error := TRUE;
           END_IF;

           //Funkcja cykliczna
           IF NOT #State.inputFlag AND NOT #State.outputFlag THEN
               IF #Reset THEN
                   #Status.ErrorStatus  := 16#0000;
                   #Status.Error := FALSE;
                       "changeState"(newState := #S_DISCONNECT,
                                     Data := #State);
               END_IF;
           END_IF;

           //Funkcja wyjściowa 
           IF #State.outputFlag THEN
               ;
           END_IF;

       #S_ENABLE_RVC:
           //Funkcja wejścia
           IF #State.inputFlag AND NOT #State.outputFlag THEN
               #State.name := 'ZEZWOLENIE NA ODBIERANIE DANYCH';
               #Connection.TRVC.ADHOC := TRUE;
               #Timers.WatchdogInitRVC.IN := TRUE;
               #Connection.TRVC.ENABLE := TRUE;
           END_IF;

           //Funkcja cykliczna
           IF NOT #State.inputFlag AND NOT #State.outputFlag THEN
               IF #Connection.TRVC.STATUS = 16#7001 OR #Connection.TRVC.STATUS = 16#7002 THEN
                   "changeState"(newState := #S_MACHINE_START,
                                 Data := #State);
               END_IF;

               IF #Timers.WatchdogInitRVC.Timer.Q THEN
                   #Status.ErrorStatus  := #E_TRCV_TIMEOUT;
                   "changeState"(newState := #S_ERROR,
                                 Data := #State);
               END_IF;
           END_IF;

           //Funkcja wyjściowa 
           IF #State.outputFlag THEN
               #Timers.WatchdogInitRVC.IN := FALSE;
           END_IF;

       #S_MACHINE_START:
           //Funkcja wejścia
           IF #State.inputFlag AND NOT #State.outputFlag THEN
               #State.name := 'TWORZENIE WIADOMOSCI';
               #MessageGenerating.len := LEN(#COMAND_SEND_MACHINE_START);
               Strg_TO_Chars(Strg := #COMAND_SEND_MACHINE_START,
                             pChars := 0,
                             Cnt => #MessageGenerating.len,
                             Chars := #MessageGenerating.chars);
               FOR #MessageGenerating.i := 0 TO #MessageGenerating.len DO
                   #Data.SEND[#MessageGenerating.i] := CHAR_TO_BYTE(#MessageGenerating.chars[#MessageGenerating.i]);
               END_FOR;
               #Connection.TSEND.LEN := DINT_TO_UDINT(#MessageGenerating.len);
               #Timers.WatchdogMachineStart.IN := TRUE;
               #Local.MessageSent := FALSE; //ZMIENNA ODPOWIADAJĄCA ZA SPRAWDZENIE CZY WIADOMOŚĆ ZOSTAŁA WYSŁANA
               #State.name := 'OCZEKIWANIE NA DANE Z KAMERY';
               #Connection.TSEND.REQ := TRUE;
           END_IF;

           //Funkcja cykliczna
           IF NOT #State.inputFlag AND NOT #State.outputFlag THEN

               //WIADOMOŚĆ POMYŚLNIE WYSŁANA
               IF #Connection.TSEND.DONE THEN
                   #Local.MessageSent := TRUE;
               END_IF;

               //ODEBRANIE WIADOMOŚCI I DEKODOWANIE
               IF #Connection.TRVC.NDR AND #Local.MessageSent THEN
                   FOR #MessageGenerating.i := 0 TO UDINT_TO_INT(#Connection.TRVC.RVC_LEN) DO
                       #MessageGenerating.chars[#MessageGenerating.i] := BYTE_TO_CHAR(#Data.RVC[#MessageGenerating.i]);
                   END_FOR;
                   Chars_TO_Strg(Chars := #MessageGenerating.chars,
                                 pChars := 0,
                                 Cnt := UDINT_TO_UINT(#Connection.TRVC.RVC_LEN),
                                 Strg => #MessageGenerating.string);
                   IF #COMMAND_RVC_MACHINE_START = #MessageGenerating.string THEN
                       "changeState"(newState := #S_IDLE,
                                     Data := #State);
                   ELSIF #COMMAND_RVC_MACHINE_START <> #MessageGenerating.string THEN
                       #Status.ErrorStatus  := #E_WRONG_RESPONSE_MACHINE_START;
                       "changeState"(newState := #S_ERROR,
                                     Data := #State);
                   END_IF;
               END_IF;

               //TIMEOUT
               IF #Timers.WatchdogMachineStart.Timer.Q THEN
   (*                //JEŚLI JUŻ BYŁY 3 PRÓBY WYSŁANIA WIADOMOŚCI
                   IF #Local.MessageSentCounter > 3 THEN
                       IF NOT #Local.MessageSent THEN
                           #Status.ErrorStatus  := #E_START_MACHINE_NOT_SENT;
                       ELSIF #Local.MessageSent THEN
                           #Status.ErrorStatus  := #E_START_MACHINE_NO_RESPONSE;
                       END_IF;
                       "changeState"(newState := #S_ERROR,
                                     Data := #State);
                       //WYSYŁANIE WIADOMOŚCI DO 3 RAZY    
                   ELSE
                       #Local.MessageSentCounter := #Local.MessageSentCounter + 1;
                       #Local.prevState := #State.state;
                       "changeState"(newState := #S_REPEAT,
                                     Data := #State);
                   END_IF; *)
                   "changeState"(newState := #S_ERROR,
                                 Data := #State);
               END_IF;
           END_IF;

           //Funkcja wyjściowa 
           IF #State.outputFlag THEN
               #Connection.TSEND.REQ := FALSE;
               #Timers.WatchdogMachineStart.IN := FALSE;
           END_IF;

       #S_IDLE:
           //Funkcja wejścia
           IF #State.inputFlag AND NOT #State.outputFlag THEN
               #Local.MessageSentCounter := 0;
               #State.name := 'OCZEKIWANIE NA WODOMIERZ';
               #Status.Busy := FALSE;
               #Status.Ready := TRUE;
               //#Status.Done := FALSE;
               #Status.Error := FALSE;
           END_IF;

           //Funkcja cykliczna
           IF NOT #State.inputFlag AND NOT #State.outputFlag THEN
               IF #Execute THEN
                    "changeState"(newState := #S_START_CAMERA,
                                 Data := #State);
               END_IF;
           END_IF;

           //Funkcja wyjściowa 
           IF #State.outputFlag THEN
               #Status.Done := FALSE;
               #Status.Ready := FALSE;
               #Status.Busy := TRUE;
           END_IF;

       #S_START_CAMERA:
           //Funkcja wejścia
           IF #State.inputFlag AND NOT #State.outputFlag THEN
               #State.name := 'WYSYLANIE DANYCH';
               #Local.MessageSent := FALSE;
               #MessageGenerating.len := LEN(#COMMAND_SEND_START_CONTROL);
               Strg_TO_Chars(Strg := #COMMAND_SEND_START_CONTROL,
                             pChars := 0,
                             Cnt => #MessageGenerating.len,
                             Chars := #MessageGenerating.chars);
               FOR #MessageGenerating.i := 0 TO #MessageGenerating.len DO
                   #Data.SEND[#MessageGenerating.i] := CHAR_TO_BYTE(#MessageGenerating.chars[#MessageGenerating.i]);
               END_FOR;
               #State.name := 'OCZEKIWANIE NA DANE Z KAMERY';
               #Connection.TSEND.LEN := DINT_TO_UDINT(#MessageGenerating.len);
               #Timers.WatchdogCamera.IN := TRUE;
               #Connection.TSEND.REQ := TRUE;
           END_IF;

           //Funkcja cykliczna
           IF NOT #State.inputFlag AND NOT #State.outputFlag THEN
               //POTWIERDZENIE WYSŁANIA WIADOMOŚCI
               IF #Connection.TSEND.DONE THEN
                   #Local.MessageSent := TRUE;
               END_IF;

               //ODEBRANIE WIADOMOŚCI I DEKODOWANIE
               IF #Connection.TRVC.NDR AND #Local.MessageSent THEN
                   FOR #MessageGenerating.i := 0 TO UDINT_TO_INT(#Connection.TRVC.RVC_LEN) DO
                       #MessageGenerating.chars[#MessageGenerating.i] := BYTE_TO_CHAR(#Data.RVC[#MessageGenerating.i]);
                   END_FOR;
                   Chars_TO_Strg(Chars := #MessageGenerating.chars,
                                 pChars := 0,
                                 Cnt := UDINT_TO_UINT(#Connection.TRVC.RVC_LEN),
                                 Strg => #MessageGenerating.string);
                   IF #COMMAND_RVC_CONTROL_DONE = #MessageGenerating.string THEN
                       #Status.Done := TRUE;
                       #DebugCounter := #DebugCounter + 1;
                       "changeState"(newState := #S_IDLE,
                                     Data := #State);
                   ELSIF #COMMAND_RVC_CONTROL_DONE <> #MessageGenerating.string THEN
                       #Status.ErrorStatus := #E_WRONG_RESPONSE_CAMERA;
                       "changeState"(newState := #S_ERROR,
                                     Data := #State);
                   END_IF; 
                   //#Status.Done := TRUE;
                   "changeState"(newState := #S_IDLE,
                                 Data := #State);
               END_IF;

               //TIMEOUT
               IF #Timers.WatchdogCamera.Timer.Q THEN
   (*                //JEŚLI JUŻ BYŁY 3 PRÓBY WYSŁANIA WIADOMOŚCI
                   IF #Local.MessageSentCounter > 3 THEN
                       IF NOT #Local.MessageSent THEN
                           #Status.ErrorStatus := #E_CAMERA_NOT_SENT;
                       ELSIF #Local.MessageSent THEN
                           #Status.ErrorStatus := #E_CAMERA_NO_RESPONSE;
                       END_IF;
                       "changeState"(newState := #S_ERROR,
                                     Data := #State);
                       //WYSYŁANIE WIADOMOŚCI DO 3 RAZY    
                   ELSE
                       #Local.MessageSentCounter := #Local.MessageSentCounter + 1;
                       #Local.prevState := #State.state;
                       "changeState"(newState := #S_REPEAT,
                                     Data := #State);
                   END_IF; 
                   "changeState"(newState := #S_ERROR,
                                 Data := #State); *)
                   "changeState"(newState := #S_ERROR,
                                 Data := #State);
               END_IF;
           END_IF;

           //Funkcja wyjściowa 
           IF #State.outputFlag THEN
               #Connection.TSEND.REQ := FALSE;
               #Timers.WatchdogCamera.IN := FALSE;
           END_IF;

       #S_REPEAT:
           "changeState"(newState := #Local.prevState,
                         Data := #State);
           //TESTOWANIE    
       #STATE_TEST:
           ;

   END_CASE;

   //GLOBAL ERRORS
   IF #Connection.TCON.ERROR THEN
       #Status.ErrorStatus := #E_TCON_ERROR;
       "changeState"(newState := #S_ERROR,
                     Data := #State);
    ELSIF #Connection.TRVC.ERROR THEN
       #Status.ErrorStatus := #E_TRCV_ERROR;
       "changeState"(newState := #S_ERROR,
                     Data := #State); 
   ELSIF #Connection.TSEND.ERROR THEN
       #Status.ErrorStatus := #E_TSEND_ERROR;
       "changeState"(newState := #S_ERROR,
                     Data := #State);
   (* ELSIF #Connection.TDISCON.ERROR THEN
       #Status.ErrorStatus := #E_TDISCON_ERROR;
       "changeState"(newState := #S_ERROR,
                     Data := #State); *)
   END_IF;

   //DISABLE FUNCTION BLOCK
   IF  #F_TRIG_Enable.Q  THEN
       "changeState"(newState := #S_DISCONNECT,
                     Data := #State);
   END_IF;

   IF #R_TRIG_Enable.Q THEN
       "changeState"(newState := #S_INITIALIZE,
                     Data := #State);
   END_IF;

   REGION Change state
       IF #State.inputFlag AND NOT #State.outputFlag THEN
           #State.inputFlag := FALSE;
       END_IF;
       #State.outputFlag := FALSE;
   END_REGION
END_REGION
END_FUNCTION_BLOCK

FUNCTION_BLOCK "ModularAxis"   // FB4, LAD
{ S7_Optimized_Access := 'TRUE' }
// stored: MemoryReserve 100, SetENOAutomatically false
   VAR_INPUT
      HomingSensor : Bool;
      Reset : Bool;
      InverterOK : Bool;
      Axis : TO_PositioningAxis;
   END_VAR
   VAR_OUTPUT
      Status : "Status";
   END_VAR
   VAR_IN_OUT
      Execute : Bool;
      PositioningAxis : "S_PositioningAxis";
   END_VAR
   VAR
      State : "s_changeState";
      Delay { S7_SetPoint := 'True'} : "s_TON";
      PowerOff { S7_SetPoint := 'True'} : "s_TON";
      MC_POWER_Instance { ExternalAccessible := 'False'; ExternalVisible := 'False'; ExternalWritable := 'False'} : MC_POWER;
      MC_RESET_Instance { ExternalAccessible := 'False'; ExternalVisible := 'False'; ExternalWritable := 'False'} : MC_RESET;
      MC_HOME_Instance { ExternalAccessible := 'False'; ExternalVisible := 'False'; ExternalWritable := 'False'} : MC_HOME;
      MC_HALT_Instance { ExternalAccessible := 'False'; ExternalVisible := 'False'; ExternalWritable := 'False'} : MC_HALT;
      MC_MOVERELATIVE_Instance { ExternalAccessible := 'False'; ExternalVisible := 'False'; ExternalWritable := 'False'} : MC_MOVERELATIVE;
      MC_MOVEJOG_Instance { ExternalAccessible := 'False'; ExternalVisible := 'False'; ExternalWritable := 'False'} : MC_MOVEJOG;
      R_TRIG_Homing { ExternalAccessible := 'False'; ExternalVisible := 'False'; ExternalWritable := 'False'} : R_TRIG;
      R_TRIG_HomeError { ExternalAccessible := 'False'; ExternalVisible := 'False'; ExternalWritable := 'False'} : R_TRIG;
      R_TRIG_HaltError { ExternalAccessible := 'False'; ExternalVisible := 'False'; ExternalWritable := 'False'} : R_TRIG;
      R_TRIG_PowerError { ExternalAccessible := 'False'; ExternalVisible := 'False'; ExternalWritable := 'False'} : R_TRIG;
      R_TRIG_JogError { ExternalAccessible := 'False'; ExternalVisible := 'False'; ExternalWritable := 'False'} : R_TRIG;
      R_TRIG_MoveRelError { ExternalAccessible := 'False'; ExternalVisible := 'False'; ExternalWritable := 'False'} : R_TRIG;
      R_TRIG_ResetError { ExternalAccessible := 'False'; ExternalVisible := 'False'; ExternalWritable := 'False'} : R_TRIG;
      F_TRIG_Inverter { ExternalAccessible := 'False'; ExternalVisible := 'False'; ExternalWritable := 'False'} : F_TRIG;
      Local : Struct
         HomingRequired : Bool;
         prevPosition : LReal;
      END_STRUCT;
   END_VAR
   VAR CONSTANT
      S_IDLE : Int := 10;
      S_HOME : Int := 20;
      S_STOP : Int := 30;
      S_ERROR : Int := 40;
      S_POWER_ON : Int := 50;
      S_MOVE_JOG : Int := 60;
      S_TEST : Int := 100;
      HOMING_ERROR : Word := 16#8000;
      HALT_ERROR : Word := 16#8001;
      POWER_ERROR : Word := 16#8002;
      JOG_ERROR : Word := 16#8003;
      MOVREL_ERROR : Word := 16#8004;
      RESET_ERROR : Word := 16#8005;
   END_VAR
BEGIN

REGION Network 1 (SCL)
   //************************************************************
   //===Author: Mateusz Połojko
   //-----Linkedin: https://pl.linkedin.com/in/mateusz-po%C5%82ojko-52a3541b1
   //-----Github: https://github.com/Bhazel95
   //===Description:
   //-----Motor control as to_speed axis
   //===Customer:
   //-----Apator Powogaz S.A.
   //************************************************************
END_REGION

REGION Network 2
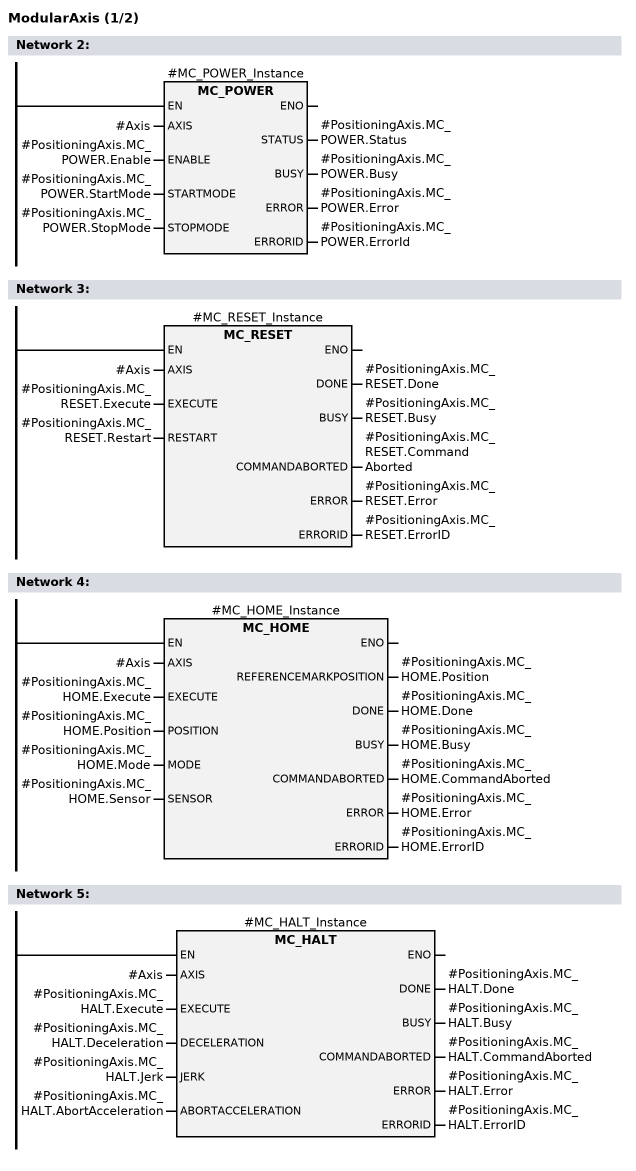
   RUNG wire#powerrail
      #MC_POWER_Instance.MC_POWER(Axis := #Axis, Enable := #PositioningAxis.MC_POWER.Enable, StartMode := #PositioningAxis.MC_POWER.StartMode, StopMode := #PositioningAxis.MC_POWER.StopMode, Status => #PositioningAxis.MC_POWER.Status, Busy => #PositioningAxis.MC_POWER.Busy, Error => #PositioningAxis.MC_POWER.Error, ErrorId => #PositioningAxis.MC_POWER.ErrorId)
   END_RUNG
   // the same network as SCL:
   #MC_POWER_Instance(Axis := #Axis,   // MC_POWER
                      Enable := #PositioningAxis.MC_POWER.Enable,
                      StartMode := #PositioningAxis.MC_POWER.StartMode,
                      StopMode := #PositioningAxis.MC_POWER.StopMode,
                      Status => #PositioningAxis.MC_POWER.Status,
                      Busy => #PositioningAxis.MC_POWER.Busy,
                      Error => #PositioningAxis.MC_POWER.Error,
                      ErrorId => #PositioningAxis.MC_POWER.ErrorId);
END_REGION

REGION Network 3
   RUNG wire#powerrail
      #MC_RESET_Instance.MC_RESET(Axis := #Axis, Execute := #PositioningAxis.MC_RESET.Execute, Restart := #PositioningAxis.MC_RESET.Restart, Done => #PositioningAxis.MC_RESET.Done, Busy => #PositioningAxis.MC_RESET.Busy, CommandAborted => #PositioningAxis.MC_RESET.CommandAborted, Error => #PositioningAxis.MC_RESET.Error, ErrorId => #PositioningAxis.MC_RESET.ErrorID)
   END_RUNG
   // the same network as SCL:
   #MC_RESET_Instance(Axis := #Axis,   // MC_RESET
                      Execute := #PositioningAxis.MC_RESET.Execute,
                      Restart := #PositioningAxis.MC_RESET.Restart,
                      Done => #PositioningAxis.MC_RESET.Done,
                      Busy => #PositioningAxis.MC_RESET.Busy,
                      CommandAborted => #PositioningAxis.MC_RESET.CommandAborted,
                      Error => #PositioningAxis.MC_RESET.Error,
                      ErrorId => #PositioningAxis.MC_RESET.ErrorID);
END_REGION

REGION Network 4
   RUNG wire#powerrail
      #MC_HOME_Instance.MC_HOME(Axis := #Axis, Execute := #PositioningAxis.MC_HOME.Execute, Position := #PositioningAxis.MC_HOME.Position, Mode := #PositioningAxis.MC_HOME.Mode, Sensor := #PositioningAxis.MC_HOME.Sensor, ReferenceMarkPosition => #PositioningAxis.MC_HOME.Position, Done => #PositioningAxis.MC_HOME.Done, Busy => #PositioningAxis.MC_HOME.Busy, CommandAborted => #PositioningAxis.MC_HOME.CommandAborted, Error => #PositioningAxis.MC_HOME.Error, ErrorId => #PositioningAxis.MC_HOME.ErrorID)
   END_RUNG
   // the same network as SCL:
   #MC_HOME_Instance(Axis := #Axis,   // MC_HOME
                     Execute := #PositioningAxis.MC_HOME.Execute,
                     Position := #PositioningAxis.MC_HOME.Position,
                     Mode := #PositioningAxis.MC_HOME.Mode,
                     Sensor := #PositioningAxis.MC_HOME.Sensor,
                     ReferenceMarkPosition => #PositioningAxis.MC_HOME.Position,
                     Done => #PositioningAxis.MC_HOME.Done,
                     Busy => #PositioningAxis.MC_HOME.Busy,
                     CommandAborted => #PositioningAxis.MC_HOME.CommandAborted,
                     Error => #PositioningAxis.MC_HOME.Error,
                     ErrorId => #PositioningAxis.MC_HOME.ErrorID);
END_REGION

REGION Network 5
   RUNG wire#powerrail
      #MC_HALT_Instance.MC_HALT(Axis := #Axis, Execute := #PositioningAxis.MC_HALT.Execute, Deceleration := #PositioningAxis.MC_HALT.Deceleration, Jerk := #PositioningAxis.MC_HALT.Jerk, AbortAcceleration := #PositioningAxis.MC_HALT.AbortAcceleration, Done => #PositioningAxis.MC_HALT.Done, Busy => #PositioningAxis.MC_HALT.Busy, CommandAborted => #PositioningAxis.MC_HALT.CommandAborted, Error => #PositioningAxis.MC_HALT.Error, ErrorId => #PositioningAxis.MC_HALT.ErrorID)
   END_RUNG
   // the same network as SCL:
   #MC_HALT_Instance(Axis := #Axis,   // MC_HALT
                     Execute := #PositioningAxis.MC_HALT.Execute,
                     Deceleration := #PositioningAxis.MC_HALT.Deceleration,
                     Jerk := #PositioningAxis.MC_HALT.Jerk,
                     AbortAcceleration := #PositioningAxis.MC_HALT.AbortAcceleration,
                     Done => #PositioningAxis.MC_HALT.Done,
                     Busy => #PositioningAxis.MC_HALT.Busy,
                     CommandAborted => #PositioningAxis.MC_HALT.CommandAborted,
                     Error => #PositioningAxis.MC_HALT.Error,
                     ErrorId => #PositioningAxis.MC_HALT.ErrorID);
END_REGION

REGION Network 6
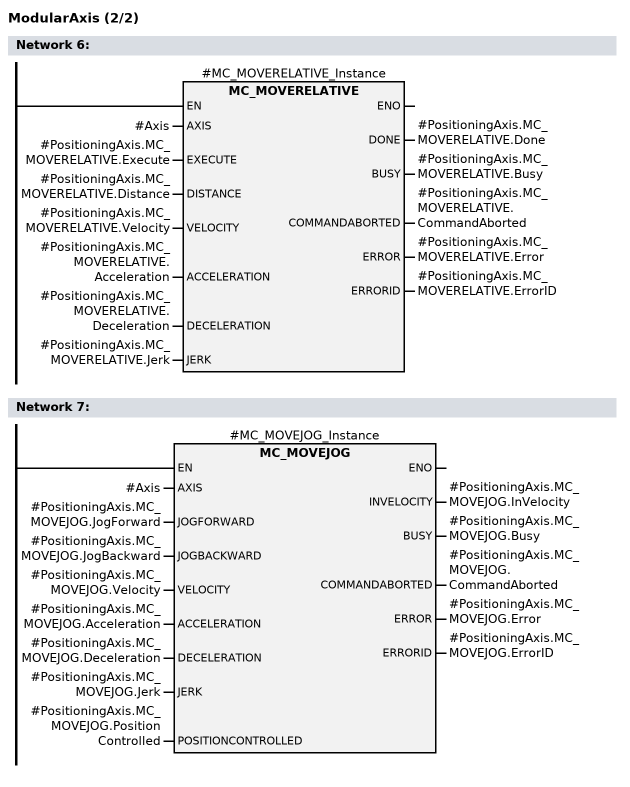
   RUNG wire#powerrail
      #MC_MOVERELATIVE_Instance.MC_MOVERELATIVE(Axis := #Axis, Execute := #PositioningAxis.MC_MOVERELATIVE.Execute, Distance := #PositioningAxis.MC_MOVERELATIVE.Distance, Velocity := #PositioningAxis.MC_MOVERELATIVE.Velocity, Acceleration := #PositioningAxis.MC_MOVERELATIVE.Acceleration, Deceleration := #PositioningAxis.MC_MOVERELATIVE.Deceleration, Jerk := #PositioningAxis.MC_MOVERELATIVE.Jerk, Done => #PositioningAxis.MC_MOVERELATIVE.Done, Busy => #PositioningAxis.MC_MOVERELATIVE.Busy, CommandAborted => #PositioningAxis.MC_MOVERELATIVE.CommandAborted, Error => #PositioningAxis.MC_MOVERELATIVE.Error, ErrorId => #PositioningAxis.MC_MOVERELATIVE.ErrorID)
   END_RUNG
   // the same network as SCL:
   #MC_MOVERELATIVE_Instance(Axis := #Axis,   // MC_MOVERELATIVE
                           Execute := #PositioningAxis.MC_MOVERELATIVE.Execute,
                           Distance := #PositioningAxis.MC_MOVERELATIVE.Distance,
                           Velocity := #PositioningAxis.MC_MOVERELATIVE.Velocity,
                           Acceleration := #PositioningAxis.MC_MOVERELATIVE.Acceleration,
                           Deceleration := #PositioningAxis.MC_MOVERELATIVE.Deceleration,
                           Jerk := #PositioningAxis.MC_MOVERELATIVE.Jerk,
                           Done => #PositioningAxis.MC_MOVERELATIVE.Done,
                           Busy => #PositioningAxis.MC_MOVERELATIVE.Busy,
                           CommandAborted => #PositioningAxis.MC_MOVERELATIVE.CommandAborted,
                           Error => #PositioningAxis.MC_MOVERELATIVE.Error,
                           ErrorId => #PositioningAxis.MC_MOVERELATIVE.ErrorID);
END_REGION

REGION Network 7
   RUNG wire#powerrail
      #MC_MOVEJOG_Instance.MC_MOVEJOG(Axis := #Axis, JogForward := #PositioningAxis.MC_MOVEJOG.JogForward, JogBackward := #PositioningAxis.MC_MOVEJOG.JogBackward, Velocity := #PositioningAxis.MC_MOVEJOG.Velocity, Acceleration := #PositioningAxis.MC_MOVEJOG.Acceleration, Deceleration := #PositioningAxis.MC_MOVEJOG.Deceleration, Jerk := #PositioningAxis.MC_MOVEJOG.Jerk, PositionControlled := #PositioningAxis.MC_MOVEJOG.PositionControlled, InVelocity => #PositioningAxis.MC_MOVEJOG.InVelocity, Busy => #PositioningAxis.MC_MOVEJOG.Busy, CommandAborted => #PositioningAxis.MC_MOVEJOG.CommandAborted, Error => #PositioningAxis.MC_MOVEJOG.Error, ErrorId => #PositioningAxis.MC_MOVEJOG.ErrorID)
   END_RUNG
   // the same network as SCL:
   #MC_MOVEJOG_Instance(Axis := #Axis,   // MC_MOVEJOG
                        JogForward := #PositioningAxis.MC_MOVEJOG.JogForward,
                        JogBackward := #PositioningAxis.MC_MOVEJOG.JogBackward,
                        Velocity := #PositioningAxis.MC_MOVEJOG.Velocity,
                        Acceleration := #PositioningAxis.MC_MOVEJOG.Acceleration,
                        Deceleration := #PositioningAxis.MC_MOVEJOG.Deceleration,
                        Jerk := #PositioningAxis.MC_MOVEJOG.Jerk,
                        PositionControlled := #PositioningAxis.MC_MOVEJOG.PositionControlled,
                        InVelocity => #PositioningAxis.MC_MOVEJOG.InVelocity,
                        Busy => #PositioningAxis.MC_MOVEJOG.Busy,
                        CommandAborted => #PositioningAxis.MC_MOVEJOG.CommandAborted,
                        Error => #PositioningAxis.MC_MOVEJOG.Error,
                        ErrorId => #PositioningAxis.MC_MOVEJOG.ErrorID);
END_REGION

REGION Network 9 (SCL)
   REGION R/F Trigs
       #F_TRIG_Inverter(CLK := #InverterOK);
       #R_TRIG_HomeError(CLK := #PositioningAxis.MC_HOME.Error);
       #R_TRIG_HaltError(CLK := #PositioningAxis.MC_HALT.Error);
       #R_TRIG_PowerError(CLK := #PositioningAxis.MC_POWER.Error);
       #R_TRIG_JogError(CLK := #PositioningAxis.MC_MOVEJOG.Error);
       #R_TRIG_MoveRelError(CLK := #PositioningAxis.MC_MOVERELATIVE.Error);
       #R_TRIG_ResetError(CLK := #PositioningAxis.MC_RESET.Error);
       #R_TRIG_Homing(CLK := #HomingSensor);

   END_REGION
   #Delay.PT := T#500MS;
   #Delay.Timer(IN := #Delay.IN,
                PT := #Delay.PT);
   #PowerOff.PT := T#180S;
   #PowerOff.Timer(IN := #PowerOff.IN,
                   PT := #PowerOff.PT);

   CASE #State.state OF
       #S_IDLE:
           //Funkcja wejścia
           IF #State.inputFlag AND NOT #State.outputFlag THEN
               #Execute := FALSE;
               #State.name := 'IDLE';
               #Status.Busy := FALSE;
               #Status.Ready := TRUE;
              // #Status.Done := FALSE;
               #Status.Error := FALSE;
               #PowerOff.IN := TRUE;
           END_IF;

           //Funkcja cykliczna
           IF NOT #State.inputFlag AND NOT #State.outputFlag THEN
               IF #PowerOff.Timer.Q THEN
                   #PositioningAxis.MC_POWER.Enable := FALSE;
               END_IF;
               IF #Reset THEN
                   // Statement section IF
                   ;
               END_IF;


               IF #Execute  THEN
                   IF #PositioningAxis.MC_POWER.Status THEN
                       #Status.Done := FALSE;
                       "changeState"(newState := #S_MOVE_JOG,
                                         Data := #State);
                   ELSE
                       #PositioningAxis.MC_POWER.Enable := FALSE;
                       "changeState"(newState := #S_POWER_ON,
                                     Data := #State);
                   END_IF;
               END_IF;
               IF #PositioningAxis.MC_MOVEJOG.JogForward OR #PositioningAxis.MC_MOVEJOG.JogBackward THEN
                   #Status.Done := FALSE;
                   #Status.Busy := TRUE;
                  //#Local.HomingRequired := TRUE;
               END_IF;
           END_IF;

           //Funkcja wyjściowa 
           IF #State.outputFlag THEN
               #PowerOff.IN := FALSE;
               #Status.Busy := TRUE;
           END_IF;

       #S_HOME:
           //Funkcja wejścia
           IF #State.inputFlag AND NOT #State.outputFlag THEN
               #State.name := 'HOMING';
               #Status.Busy := TRUE;
               #Status.Ready := FALSE;
               #Status.Done := FALSE;
               #Status.Error := FALSE;
               #PositioningAxis.MC_HOME.Mode := 8;
               #PositioningAxis.MC_HOME.Execute := TRUE;
           END_IF;

           //Funkcja cykliczna
           IF NOT #State.inputFlag AND NOT #State.outputFlag THEN
               IF #PositioningAxis.MC_HOME.Done THEN
                   #Local.HomingRequired := FALSE;
                   #Status.Done := TRUE;
                   "changeState"(newState := #S_IDLE,
                                 Data := #State);
               END_IF;
           END_IF;

           //Funkcja wyjściowa 
           IF #State.outputFlag THEN
               #PositioningAxis.MC_HOME.Execute := FALSE;
           END_IF;

       #S_ERROR:
           //Funkcja wejścia
           IF #State.inputFlag AND NOT #State.outputFlag THEN
               #State.name := 'ERROR';
               #Status.Busy := FALSE;
               #Status.Ready := FALSE;
               //#Status.Done := FALSE;
               #Status.Error := TRUE;
             //#Local.HomingRequired := TRUE;
               #PositioningAxis.MC_HOME.Execute := FALSE;
               #PositioningAxis.MC_POWER.Enable := FALSE;
               #PositioningAxis.MC_MOVERELATIVE.Execute := FALSE;
               #PositioningAxis.MC_HALT.Execute := FALSE;
               #PositioningAxis.MC_RESET.Execute := FALSE;
               #PositioningAxis.MC_MOVEJOG.JogBackward := FALSE;
               #PositioningAxis.MC_MOVEJOG.JogForward := FALSE;
           END_IF;

           //Funkcja cykliczna
           IF NOT #State.inputFlag AND NOT #State.outputFlag THEN
               IF #Reset THEN
                  // #MC_RESET_Instance.Restart := FALSE;
                   #PositioningAxis.MC_RESET.Execute := TRUE;
               END_IF;
               IF #PositioningAxis.MC_RESET.Done AND #InverterOK THEN
                   "changeState"(newState := #S_POWER_ON,
                                 Data := #State);
               END_IF;
           END_IF;

           //Funkcja wyjściowa 
           IF #State.outputFlag THEN
               #Status.Error := FALSE;
               #Status.Busy := TRUE;
               #PositioningAxis.MC_RESET.Execute := FALSE;
           END_IF;

       #S_POWER_ON:
           //Funkcja wejścia
           IF #State.inputFlag AND NOT #State.outputFlag THEN
               #State.name := 'ERROR';
               #Status.Busy := TRUE;
               #Status.Ready := FALSE;
               #Status.Done := FALSE;
               #Status.Error := FALSE;
               #PositioningAxis.MC_POWER.Enable := TRUE;
           END_IF;

           //Funkcja cykliczna
           IF NOT #State.inputFlag AND NOT #State.outputFlag THEN
               IF #PositioningAxis.MC_POWER.Status THEN
                   "changeState"(newState := #S_IDLE,
                                 Data := #State);
               END_IF;
           END_IF;

           //Funkcja wyjściowa 
           IF #State.outputFlag THEN
               ;
           END_IF;

       #S_MOVE_JOG:
           //Funkcja wejścia
           IF #State.inputFlag AND NOT #State.outputFlag THEN
               #State.name := 'MOVING';
               #Status.Busy := TRUE;
               #Status.Ready := FALSE;
               #Status.Done := FALSE;
               #Status.Error := FALSE;
               #Local.prevPosition := #Axis.ActualPosition;
               #PositioningAxis.MC_MOVEJOG.Acceleration := 60;
               #PositioningAxis.MC_MOVEJOG.Deceleration := 120;
               #PositioningAxis.MC_MOVEJOG.Velocity := 50;
               #PositioningAxis.MC_MOVEJOG.JogBackward := FALSE;
               #PositioningAxis.MC_MOVEJOG.JogForward := TRUE;
               #Delay.IN := FALSE;
           END_IF;

           //Funkcja cykliczna
           IF NOT #State.inputFlag AND NOT #State.outputFlag THEN
               IF #R_TRIG_Homing.Q THEN
                   #Status.Done := TRUE;
                   #PositioningAxis.MC_MOVEJOG.JogBackward := FALSE;
                   #PositioningAxis.MC_MOVEJOG.JogForward := FALSE;
                   #Delay.IN := TRUE;
               END_IF;
               IF #Delay.Timer.Q THEN
                   "changeState"(newState := #S_IDLE,
                                 Data := #State);
               END_IF;

           END_IF;

           //Funkcja wyjściowa 
           IF #State.outputFlag THEN
               #Delay.IN := FALSE;
           END_IF;

       #S_TEST:
           ;
   END_CASE;

   IF #R_TRIG_HomeError.Q THEN
       #Status.ErrorStatus := #HOMING_ERROR;
       "changeState"(newState := #S_ERROR,
                     Data := #State);
   ELSIF #R_TRIG_HaltError.Q THEN
       #Status.ErrorStatus := #HALT_ERROR;
       "changeState"(newState := #S_ERROR,
                     Data := #State);
   ELSIF #R_TRIG_JogError.Q THEN
       #Status.ErrorStatus := #JOG_ERROR;
       "changeState"(newState := #S_ERROR,
                     Data := #State);
   ELSIF #R_TRIG_MoveRelError.Q THEN
       #Status.ErrorStatus := #MOVREL_ERROR;
       "changeState"(newState := #S_ERROR,
                     Data := #State);
   ELSIF #R_TRIG_PowerError.Q THEN
       #Status.ErrorStatus := #POWER_ERROR;
       "changeState"(newState := #S_ERROR,
                     Data := #State);
   ELSIF #R_TRIG_ResetError.Q THEN
       #Status.ErrorStatus := #RESET_ERROR;
       "changeState"(newState := #S_ERROR,
                     Data := #State);
   END_IF;

   IF #F_TRIG_Inverter.Q THEN
       "changeState"(newState := #S_ERROR,
                     Data := #State);
   END_IF;

   IF NOT "DEV_7".Convoyer.Modular_A.Sensors.JogBack THEN
       #PositioningAxis.MC_MOVEJOG.JogBackward := FALSE;
   END_IF;

   REGION Change state
       IF #State.inputFlag AND NOT #State.outputFlag THEN
           #State.inputFlag := FALSE;
       END_IF;
       #State.outputFlag := FALSE;
   END_REGION
END_REGION
END_FUNCTION_BLOCK

FUNCTION_BLOCK "Blow"
{ S7_Optimized_Access := 'TRUE' }
VERSION : 0.1
   VAR_INPUT 
      "Timer" : Time;
   END_VAR

   VAR_IN_OUT 
      Execute : Bool;
      Coil : Bool;
   END_VAR

   VAR 
      Blow { S7_SetPoint := 'False'} : "s_TON";
      R_TRIG_Exe {InstructionName := 'R_TRIG'; LibVersion := '1.0'; ExternalAccessible := 'False'; ExternalVisible := 'False'; ExternalWritable := 'False'; S7_SetPoint := 'False'} : R_TRIG;
      R_TRIG_Done {InstructionName := 'R_TRIG'; LibVersion := '1.0'; ExternalAccessible := 'False'; ExternalVisible := 'False'; ExternalWritable := 'False'; S7_SetPoint := 'False'} : R_TRIG;
   END_VAR


BEGIN
	REGION r trigs
	    #R_TRIG_Exe(CLK := #Execute);
	    #R_TRIG_Done(CLK := #Blow.Timer.Q);
	END_REGION
	
	
	    #Blow.PT := #Timer;
	    #Blow.IN := #Execute;
	    #Blow.Timer(IN := #Blow.IN,
	                PT := #Blow.PT);
	    
	    IF #R_TRIG_Exe.Q THEN
	        #Coil := TRUE;
	    END_IF;
	    IF #R_TRIG_Done.Q THEN
	        #Coil := FALSE;
	        #Execute := FALSE;
	    END_IF;
	    
	    
	    
	    
	
END_FUNCTION_BLOCK

FUNCTION_BLOCK "ModularConvoyer_Speed"
{ S7_Optimized_Access := 'TRUE' }
VERSION : 0.1
   VAR_INPUT 
      Axis {InstructionName := 'TO_SpeedAxis'; LibVersion := '7.0'} : TO_SpeedAxis;
   END_VAR

   VAR_IN_OUT 
      Convoyer : "Modular_SPEED";
      Diagnostic : "DiagnosticMainCabinet";
      ProducedUnits : DInt;
   END_VAR

   VAR 
      R_TRIG_CriticalError {InstructionName := 'R_TRIG'; LibVersion := '1.0'; ExternalAccessible := 'False'; ExternalVisible := 'False'; ExternalWritable := 'False'; S7_SetPoint := 'False'} : R_TRIG;
      R_TRIG_StampingDone {InstructionName := 'R_TRIG'; LibVersion := '1.0'; ExternalAccessible := 'False'; ExternalVisible := 'False'; ExternalWritable := 'False'; S7_SetPoint := 'False'} : R_TRIG;
      R_TRIG_CameraDone {InstructionName := 'R_TRIG'; LibVersion := '1.0'; ExternalAccessible := 'False'; ExternalVisible := 'False'; ExternalWritable := 'False'; S7_SetPoint := 'False'} : R_TRIG;
      R_TRIG_SortingDone {InstructionName := 'R_TRIG'; LibVersion := '1.0'; ExternalAccessible := 'False'; ExternalVisible := 'False'; ExternalWritable := 'False'; S7_SetPoint := 'False'} : R_TRIG;
      R_TRIG_ConvoyerDone {InstructionName := 'R_TRIG'; LibVersion := '1.0'; ExternalAccessible := 'False'; ExternalVisible := 'False'; ExternalWritable := 'False'; S7_SetPoint := 'False'} : R_TRIG;
      R_TRIG_Stop {InstructionName := 'R_TRIG'; LibVersion := '1.0'; ExternalAccessible := 'False'; ExternalVisible := 'False'; ExternalWritable := 'False'; S7_SetPoint := 'False'} : R_TRIG;
      State { S7_SetPoint := 'False'} : "s_changeState";
      Local : Struct
         AutoMode : Bool;
         Buttons : Struct
            START : Bool;
            RESET : Bool;
            STOP : Bool;
         END_STRUCT;
         PermissionToStart : Bool;
         PermissionGoBack : Bool;
         ActionDone : Struct
            Stamping : Bool;
            Camera : Bool;
            Sorting : Bool;
         END_STRUCT;
         Execute : Struct
            Stamping : Bool;
            Camera : Bool;
            Sorting : Bool;
            Convoyer : Bool;
            Blow : Bool;
         END_STRUCT;
         ActionToDo : Struct
            Stamping : Bool;
            Camera : Bool;
            Blow : Bool;
            PreCamera : Array[0..1] of Bool;
         END_STRUCT;
         DoubleStampingDone : Bool;
         StampingTime : Time;
         isMoved : Bool;
         backwardProcess : Bool;
      END_STRUCT;
      Timers : Struct
         WatchdogGoModules { S7_SetPoint := 'False'} : "s_TON";
         WatchdogGoConvoyer : "s_TON";
         Delay : "s_TON";
         DoubleStamp : "s_TON";
         UnloadTimer {InstructionName := 'TON_TIME'; LibVersion := '1.0'; ExternalAccessible := 'False'; ExternalVisible := 'False'; ExternalWritable := 'False'; S7_SetPoint := 'False'} : TON_TIME;
         OskarDelay : "s_TON";
         GoBackwardEnable : "s_TON";
         GoBackward : "s_TON";
      END_STRUCT;
      CameraConnectionTCP_Instance { ExternalAccessible := 'False'; ExternalVisible := 'False'; ExternalWritable := 'False'; S7_SetPoint := 'False'} : "CameraConnectionTCP";
      PositioningAxis_Instance { ExternalAccessible := 'False'; ExternalVisible := 'False'; ExternalWritable := 'False'; S7_SetPoint := 'False'} : "ModularAxis_Speed";
      Blow_Instance : "Blow";
      Stamping_Instance : "Stamping";
   END_VAR

   VAR CONSTANT 
      S_IDLE : Int := 0;
      S_ERROR : Int := 20;
      S_GO_CONVOYER : Int := 30;
      S_GO_MODULES : Int := 40;
      S_GO_BACK : Int := 50;
      TEST : Int := 100;
      E_MODULES_TIMEOUT : Word := 16#8000;
      E_CONVOYER_TIMEOUT : Word := 16#8001;
   END_VAR


BEGIN
	//************************************************************
	//===Author: Mateusz Połojko
	//-----Linkedin: https://pl.linkedin.com/in/mateusz-po%C5%82ojko-52a3541b1
	//-----Github: https://github.com/Bhazel95
	//===Description:
	//-----Main function block for convoyer + executive modules control
	//===Customer:
	//-----Apator Powogaz S.A.
	//************************************************************
	
	REGION R/F_TRIG
	    #R_TRIG_CriticalError(CLK := NOT #Convoyer.Safety.SafetyOK OR #PositioningAxis_Instance.Status.Error);
	    #R_TRIG_StampingDone(CLK := #Stamping_Instance.Status.Done);
	    #R_TRIG_CameraDone(CLK := #CameraConnectionTCP_Instance.Status.Done);
	    #R_TRIG_SortingDone(CLK := #Convoyer.SortingStatus.Done);
	    #R_TRIG_ConvoyerDone(CLK := #PositioningAxis_Instance.Status.Ready);
	    #R_TRIG_Stop(CLK := #Local.Buttons.STOP AND #Local.AutoMode);
	END_REGION
	
	REGION Timers
	    //WATCHDOG MACHINE START
	    #Timers.WatchdogGoModules.PT := T#15S;
	    #Timers.WatchdogGoModules.Timer(IN := #Timers.WatchdogGoModules.IN,
	                                    PT := #Timers.WatchdogGoModules.PT);
	    #Timers.WatchdogGoConvoyer.PT := T#10S;
	    #Timers.WatchdogGoConvoyer.Timer(IN := #Timers.WatchdogGoConvoyer.IN,
	                                     PT := #Timers.WatchdogGoConvoyer.PT);
	    #Timers.Delay.PT := T#7S;
	    #Timers.Delay.Timer(IN := #Timers.Delay.IN,
	                        PT := #Timers.Delay.PT);
	    
	    #Timers.DoubleStamp.PT := T#500MS;
	    #Timers.DoubleStamp.Timer(IN := #Timers.DoubleStamp.IN,
	                              PT := #Timers.DoubleStamp.PT);
	    
	    #Timers.OskarDelay.PT := T#5000MS;
	    #Timers.OskarDelay.Timer(IN := #Timers.OskarDelay.IN,
	                             PT := #Timers.OskarDelay.PT);
	    
	    #Timers.GoBackwardEnable.PT := T#3000MS;
	    #Timers.GoBackwardEnable.Timer(IN := #Convoyer.ButtonControl.ButtonBoxLeft.ButtonReset OR #Convoyer.ButtonControl.ButtonBoxRight.ButtonReset,
	                                   PT := #Timers.GoBackwardEnable.PT);
	    
	    #Timers.GoBackward.PT := T#2000MS;
	    #Timers.GoBackward.Timer(IN := #Timers.GoBackward.IN,
	                             PT := #Timers.GoBackward.PT);
	    
	    #Timers.UnloadTimer(IN := NOT #Convoyer.Sensors.UnloadingPresence,
	                        PT := T#1000MS);
	END_REGION
	
	//Permission to start
	#Local.PermissionToStart := #Diagnostic.DiagnosticOK AND NOT #Convoyer.Alarms.Fault24V AND #Convoyer.Safety.SafetyOK
	AND NOT #Convoyer.Alarms.Present AND #Convoyer.Pneumatics.Stamping.Sensors.In AND #Convoyer.Safety.LightCurtain_Stamping
	AND NOT #Convoyer.Pneumatics.Stamping.Sensors.Out AND (#Convoyer.CameraStatus.Ready OR NOT #Convoyer.HMI.Camera.Enable)
	AND #Convoyer.MotorStatus.Ready AND #Convoyer.Sensors.Stamp_Check_1 AND #Convoyer.Sensors.UnloadingPresence AND #Convoyer.Sensors.Span;
	
	#Local.PermissionGoBack := #Diagnostic.DiagnosticOK AND #Convoyer.Safety.SafetyOK
	AND NOT #Convoyer.Alarms.Present AND #Convoyer.Pneumatics.Stamping.Sensors.In
	AND NOT #Convoyer.Pneumatics.Stamping.Sensors.Out AND #Convoyer.MotorStatus.Ready AND #Convoyer.Sensors.Stamp_Check_1 AND #Convoyer.Sensors.UnloadingPresence AND #Convoyer.Sensors.Span AND #Convoyer.Sensors.JogBack;
	
	//Start button
	#Local.Buttons.START := #Convoyer.ButtonControl.ButtonBoxLeft.ButtonStart OR #Convoyer.ButtonControl.ButtonBoxRight.ButtonStart OR #Convoyer.HMI.Buttons.Start;
	//Stop button
	#Local.Buttons.STOP := #Convoyer.ButtonControl.ButtonBoxLeft.ButtonStop OR #Convoyer.ButtonControl.ButtonBoxRight.ButtonStop OR #Convoyer.HMI.Buttons.Stop;
	//Reset button
	#Local.Buttons.RESET := #Convoyer.ButtonControl.ButtonBoxLeft.ButtonReset OR #Convoyer.ButtonControl.ButtonBoxRight.ButtonReset OR #Convoyer.ButtonControl.CabinetBox.ButtonReset;
	
	CASE #State.state OF
	    #S_IDLE:
	        //Funkcja wejścia
	        IF #State.inputFlag AND NOT #State.outputFlag THEN
	            #Convoyer.ConvoyerStatus.Busy := FALSE;
	            #Convoyer.ConvoyerStatus.Done := FALSE;
	            #Convoyer.ConvoyerStatus.Error := FALSE;
	            #Convoyer.ConvoyerStatus.ErrorStatus := 16#0000;
	            #Convoyer.ConvoyerStatus.Ready := TRUE;
	        END_IF;
	        
	        //Funkcja cykliczna
	        IF NOT #State.inputFlag AND NOT #State.outputFlag THEN
	            //ZABEZPIECZENIE PRZED MANUALNYM RUSZENIEM TRANSPORTERA
	            IF #Convoyer.MotorControl.MC_MOVEJOG.JogBackward OR #Convoyer.MotorControl.MC_MOVEJOG.JogForward THEN
	                #Local.isMoved := TRUE;
	            END_IF;
	            IF #Convoyer.Safety.LightCurtain_Stamping AND #Local.PermissionToStart AND (#Local.Buttons.START OR #Local.AutoMode) AND NOT #Local.Buttons.STOP AND NOT #Local.Buttons.RESET THEN
	                #Local.AutoMode := TRUE;
	                IF ((NOT #Convoyer.Sensors.StampingPresence AND NOT #Local.ActionDone.Stamping) OR (NOT #Convoyer.Sensors.CameraPresence AND NOT #Local.ActionDone.Camera)) AND NOT #Local.isMoved THEN
	                    "changeState"(newState := #S_GO_MODULES,
	                                  Data := #State);
	                ELSIF ((#Local.ActionDone.Stamping OR #Convoyer.Sensors.StampingPresence) AND (#Local.ActionDone.Camera OR #Convoyer.Sensors.CameraPresence)) OR #Local.isMoved THEN
	                    "changeState"(newState := #S_GO_CONVOYER,
	                                  Data := #State);
	                END_IF;
	            END_IF;
	            //COFANIE TRANSPORTERA
	            IF NOT #Local.AutoMode AND #Local.PermissionGoBack AND #Timers.GoBackwardEnable.Timer.Q AND NOT #Local.Buttons.START AND NOT #Local.Buttons.STOP THEN
	                #Local.isMoved := TRUE;
	                "changeState"(newState := #S_GO_BACK,
	                              Data := #State);
	            END_IF;
	            
	        END_IF;
	        
	        //Funkcja wyjściowa 
	        IF #State.outputFlag THEN
	            #Convoyer.ConvoyerStatus.Ready := FALSE;
	            #Convoyer.ConvoyerStatus.Busy := TRUE;
	        END_IF;
	        
	    #S_ERROR:
	        //Funkcja wejścia
	        IF #State.inputFlag AND NOT #State.outputFlag THEN
	            #Convoyer.ConvoyerStatus.Busy := FALSE;
	            #Convoyer.ConvoyerStatus.Done := FALSE;
	            #Convoyer.ConvoyerStatus.Error := TRUE;
	            #Convoyer.ConvoyerStatus.Ready := FALSE;
	            #Timers.WatchdogGoConvoyer.IN := FALSE;
	            #Timers.WatchdogGoModules.IN := FALSE;
	            #Local.Execute.Convoyer := FALSE;
	            #Local.Execute.Stamping := FALSE;
	            #Local.Execute.Camera := FALSE;
	            //#Local.ActionDone.Camera := FALSE;
	            #Local.AutoMode := FALSE;
	        END_IF;
	        
	        //Funkcja cykliczna
	        IF NOT #State.inputFlag AND NOT #State.outputFlag THEN
	            IF #Local.Buttons.RESET AND NOT #Convoyer.Alarms.Present AND #Convoyer.Safety.SafetyOK
	                AND (#CameraConnectionTCP_Instance.Status.Ready OR NOT #Convoyer.HMI.Camera.Enable) AND #PositioningAxis_Instance.Status.Ready
	                AND (#Stamping_Instance.Status.Ready OR NOT #Convoyer.HMI.Stamping.Enable) AND #Local.PermissionToStart THEN
	                #Convoyer.ConvoyerStatus.Error := FALSE;
	                "changeState"(newState := #S_IDLE,
	                              Data := #State);
	            END_IF;
	        END_IF;
	        
	        //Funkcja wyjściowa 
	        IF #State.outputFlag THEN
	            ;
	        END_IF;
	        
	    #S_GO_CONVOYER:
	        //Funkcja wejścia
	        IF #State.inputFlag AND NOT #State.outputFlag THEN
	            #Timers.WatchdogGoConvoyer.IN := TRUE;
	            #Local.ActionDone.Stamping := FALSE;
	            #Local.ActionDone.Camera := FALSE;
	            #Local.ActionDone.Sorting := FALSE;
	            #Local.ActionToDo.PreCamera[1] := #Local.ActionToDo.PreCamera[0];
	            #Local.Execute.Convoyer := TRUE;
	        END_IF;
	        
	        //Funkcja cykliczna
	        IF NOT #State.inputFlag AND NOT #State.outputFlag THEN
	            IF #R_TRIG_ConvoyerDone.Q THEN
	                #Local.isMoved := FALSE;
	                IF NOT #Local.AutoMode OR NOT #Convoyer.Safety.LightCurtain_Stamping THEN
	                    "changeState"(newState := #S_IDLE,
	                                  Data := #State);
	                ELSE
	                    "changeState"(newState := #S_GO_MODULES,
	                                  Data := #State);
	                END_IF;
	            END_IF;
	            IF #PositioningAxis_Instance.Status.Error THEN
	                "changeState"(newState := #S_ERROR,
	                              Data := #State);
	            END_IF;
	            //WATCHDOG
	            IF #Timers.WatchdogGoConvoyer.Timer.Q THEN
	                #PositioningAxis_Instance.Status.ErrorStatus := #E_CONVOYER_TIMEOUT;
	                "changeState"(newState := #S_ERROR,
	                              Data := #State);
	            END_IF;
	        END_IF;
	        
	        //Funkcja wyjściowa 
	        IF #State.outputFlag THEN
	            #Local.Execute.Convoyer := FALSE;
	            #Local.ActionDone.Stamping := FALSE;
	            #Local.ActionDone.Camera := FALSE;
	            #Local.ActionDone.Sorting := FALSE;
	            #Timers.WatchdogGoConvoyer.IN := FALSE;
	            #Local.Execute.Convoyer := FALSE;
	        END_IF;
	        
	    #S_GO_MODULES:
	        //Funkcja wejścia
	        IF #State.inputFlag AND NOT #State.outputFlag THEN
	            #Timers.OskarDelay.IN := TRUE;
	            #Timers.WatchdogGoModules.IN := TRUE;
	            #Timers.Delay.IN := TRUE;
	            #Local.DoubleStampingDone := FALSE;
	            IF #Convoyer.HMI.Stamping.Double THEN
	                #Local.StampingTime := T#1MS;
	            ELSE
	                #Local.StampingTime := #Convoyer.HMI.Stamping.TimerStamping;
	            END_IF;
	            #Local.Execute.Blow := #Convoyer.Sensors.BlowPresence AND #Convoyer.HMI.Blow.Enable;
	            #Local.Execute.Stamping := NOT #Local.ActionDone.Stamping AND NOT #Convoyer.Sensors.StampingPresence AND #Convoyer.HMI.Stamping.Enable;
	            
	            //TUTAJ NA DOLE
	            #Local.Execute.Camera := ((NOT #Local.ActionDone.Camera AND NOT #Convoyer.Sensors.CameraPresence) OR (#Local.ActionToDo.PreCamera[1] AND NOT #Local.ActionDone.Camera)) AND #Convoyer.HMI.Camera.Enable;
	            #Local.ActionToDo.Stamping := #Local.Execute.Stamping;
	            #Local.ActionToDo.Camera := #Local.Execute.Camera;
	            #Local.ActionToDo.PreCamera[0] := #Convoyer.Sensors.BlowPresence; //DODANE ABY ZOBACZYC CZY WYELIMINUJE BLAD BRAKU ZDJEC
	        END_IF;
	        //Funkcja cykliczna
	        IF NOT #State.inputFlag AND NOT #State.outputFlag THEN
	            REGION double stamping
	                IF #Convoyer.HMI.Stamping.Double AND NOT #Local.DoubleStampingDone AND #Timers.DoubleStamp.Timer.Q THEN
	                    #Local.StampingTime := #Convoyer.HMI.Stamping.TimerStamping;
	                    #Local.DoubleStampingDone := TRUE;
	                    #Local.Execute.Stamping := TRUE;
	                END_IF;
	            END_REGION
	            
	            IF #R_TRIG_CameraDone.Q THEN
	                #Local.ActionDone.Camera := TRUE;
	                #Local.ActionToDo.Camera := FALSE;
	                #Local.Execute.Camera := FALSE;
	            END_IF;
	            IF #R_TRIG_SortingDone.Q THEN
	                #Local.ActionDone.Sorting := TRUE;
	            END_IF;
	            IF #R_TRIG_StampingDone.Q THEN
	                #ProducedUnits := #ProducedUnits + 1;
	                IF NOT #Convoyer.HMI.Stamping.Double THEN
	                    #Local.ActionDone.Stamping := TRUE;
	                    #Local.ActionToDo.Stamping := FALSE;
	                    #Local.Execute.Stamping := FALSE;
	                ELSIF #Convoyer.HMI.Stamping.Double AND NOT #Local.DoubleStampingDone THEN
	                    #Timers.DoubleStamp.IN := TRUE;
	                    #Local.Execute.Stamping := FALSE;
	                ELSIF #Convoyer.HMI.Stamping.Double AND #Local.DoubleStampingDone THEN
	                    #Local.ActionDone.Stamping := TRUE;
	                    #Local.ActionToDo.Stamping := FALSE;
	                    #Local.Execute.Stamping := FALSE;
	                END_IF;
	            END_IF;
	            
	            //Oczekiwanie na potwierdzenia blokow  - komentarz -->> opoznienie zalaczenia ruchu stolu dla Oskara
	            IF (#Local.ActionDone.Stamping OR NOT #Local.ActionToDo.Stamping) AND (#Local.ActionDone.Camera OR NOT #Local.ActionToDo.Camera) AND NOT #Local.Execute.Blow (* AND #Timers.OskarDelay.Timer.Q *)THEN
	                IF NOT #Local.AutoMode THEN
	                    "changeState"(newState := #S_IDLE,
	                                  Data := #State);
	                ELSE
	                    IF #Local.PermissionToStart THEN
	                        "changeState"(newState := #S_GO_CONVOYER,
	                                      Data := #State);
	                    ELSE
	                        "changeState"(newState := #S_IDLE,
	                                      Data := #State);
	                    END_IF;
	                END_IF;
	            END_IF;
	            //Modules Error
	            IF (#CameraConnectionTCP_Instance.Status.Error OR #Stamping_Instance.Status.Error) AND #Timers.Delay.Timer.Q THEN
	                "changeState"(newState := #S_ERROR,
	                              Data := #State);
	            END_IF;
	            
	            //WATCHDOG
	            IF #Timers.WatchdogGoModules.Timer.Q THEN
	                #PositioningAxis_Instance.Status.ErrorStatus := #E_MODULES_TIMEOUT;
	                "changeState"(newState := #S_ERROR,
	                              Data := #State);
	            END_IF;
	        END_IF;
	        
	        //Funkcja wyjściowa 
	        IF #State.outputFlag THEN
	            #Timers.Delay.IN := FALSE;
	            #Timers.OskarDelay.IN := FALSE;
	            #Timers.DoubleStamp.IN := FALSE;
	            #Timers.WatchdogGoModules.IN := FALSE;
	            #Local.Execute.Stamping := FALSE;
	            #Local.Execute.Camera := FALSE;
	            #Local.Execute.Sorting := FALSE;
	        END_IF;
	        
	    #S_GO_BACK:
	        //Funkcja wejścia
	        IF #State.inputFlag AND NOT #State.outputFlag THEN
	            #Local.backwardProcess := TRUE;
	            #Timers.GoBackward.IN := TRUE;
	            #Local.isMoved := TRUE;
	            #Convoyer.MotorControl.MC_MOVEJOG.JogBackward := TRUE;
	            
	        END_IF;
	        
	        //Funkcja cykliczna
	        IF NOT #State.inputFlag AND NOT #State.outputFlag THEN
	            IF (#Timers.GoBackward.Timer.Q AND #Convoyer.Safety.LightCurtain_Stamping) OR NOT #Convoyer.Sensors.JogBack THEN
	                #Convoyer.MotorControl.MC_MOVEJOG.JogBackward := FALSE;
	                "changeState"(newState := #S_IDLE,
	                              Data := #State);
	            END_IF;
	        END_IF;
	        
	        //Funkcja wyjściowa 
	        IF #State.outputFlag THEN
	            #Local.backwardProcess := FALSE;
	            #Convoyer.MotorControl.MC_MOVEJOG.JogBackward := FALSE;
	            #Timers.GoBackward.IN := FALSE;
	        END_IF;
	        
	END_CASE;
	
	REGION FunctionBlocks
	    #Stamping_Instance(Reset := #Local.Buttons.RESET,
	                       SecondPush := #Convoyer.HMI.Stamping.SecondPush,
	                       TimerSecondPush := #Convoyer.HMI.Stamping.TimerSecond,
	                       PreasureSecondPush := #Convoyer.HMI.Stamping.SecondPreasure,
	                       TimerStamp := #Convoyer.HMI.Stamping.TimerStamping,
	                       TimerMax := #Convoyer.HMI.Stamping.TimerMaxPreasure,
	                       MaxPreasure := #Convoyer.HMI.Stamping.MaxPreasure,
	                       RegularPreasure := #Convoyer.HMI.Stamping.RegularPreasure,
	                       Status => #Convoyer.StampingStatus,
	                       Valve := #Convoyer.Pneumatics.Stamping,
	                       ITV := #Convoyer.Pneumatics.IVT,
	                       Execute := #Local.Execute.Stamping);
	    #CameraConnectionTCP_Instance(Enable := #Convoyer.HMI.Camera.Enable,
	                                  Execute := #Local.Execute.Camera,
	                                  Reset := #Local.Buttons.RESET,
	                                  ConnectionTimer := #Convoyer.HMI.Camera.TimerConnection,
	                                  Status => #Convoyer.CameraStatus,
	                                  Parameters := #Convoyer.CameraConnection);
	    #PositioningAxis_Instance(HomingSensor := #Convoyer.Sensors.Homing_I,
	                              Reset := #Local.Buttons.RESET,
	                              InverterOK := #Convoyer.Safety.InverterOK,
	                              Axis := #Axis,
	                              Status => #Convoyer.MotorStatus,
	                              Execute := #Local.Execute.Convoyer,
	                              PositioningAxis := #Convoyer.MotorControl);
	    #Blow_Instance(Timer := #Convoyer.HMI.Blow."Time",
	                   Execute := #Local.Execute.Blow,
	                   Coil := #Convoyer.Pneumatics.Valve.Coils.Out);
	END_REGION
	
	REGION Lights
	    //RESET BUTTON
	    #Convoyer.ButtonControl.ButtonBoxLeft.LightReset := #Convoyer.ConvoyerStatus.Error OR #Convoyer.CameraStatus.Error OR #Convoyer.StampingStatus.Error OR #Convoyer.MotorStatus.Error OR (NOT #Convoyer.Pneumatics.Stamping.Sensors.In AND #Convoyer.StampingStatus.Ready) OR (#Local.backwardProcess AND "Clock_1Hz");
	    #Convoyer.ButtonControl.ButtonBoxRight.LightReset := #Convoyer.ConvoyerStatus.Error OR #Convoyer.CameraStatus.Error OR #Convoyer.StampingStatus.Error OR #Convoyer.MotorStatus.Error OR (NOT #Convoyer.Pneumatics.Stamping.Sensors.In AND #Convoyer.StampingStatus.Ready) OR (#Local.backwardProcess AND "Clock_1Hz");
	    #Convoyer.ButtonControl.CabinetBox.LightReset := #Convoyer.ConvoyerStatus.Error OR #Convoyer.CameraStatus.Error OR #Convoyer.StampingStatus.Error OR #Convoyer.MotorStatus.Error OR (NOT #Convoyer.Pneumatics.Stamping.Sensors.In AND #Convoyer.StampingStatus.Ready);
	    //STOP BUTTON
	    #Convoyer.ButtonControl.ButtonBoxLeft.LightStop := #Convoyer.ConvoyerStatus.Busy AND NOT #Local.AutoMode;
	    #Convoyer.ButtonControl.ButtonBoxRight.LightStop := #Convoyer.ConvoyerStatus.Busy AND NOT #Local.AutoMode;
	    //START BUTTON
	    #Convoyer.ButtonControl.ButtonBoxLeft.LightStart := #Convoyer.ConvoyerStatus.Ready AND #Local.PermissionToStart AND NOT #Local.AutoMode;
	    #Convoyer.ButtonControl.ButtonBoxRight.LightStart := #Convoyer.ConvoyerStatus.Ready AND #Local.PermissionToStart AND NOT #Local.AutoMode;
	    //ANDON 
	    #Convoyer.Lights.Red := #Convoyer.ConvoyerStatus.Error OR #Convoyer.CameraStatus.Error OR #Convoyer.StampingStatus.Error OR #Convoyer.MotorStatus.Error;
	    #Convoyer.Lights.Green := #Convoyer.ConvoyerStatus.Busy OR #Local.AutoMode;
	    #Convoyer.Lights.Blue := #Convoyer.ConvoyerStatus.Ready AND #Local.PermissionToStart AND NOT #Local.AutoMode;
	    #Convoyer.Lights.Orange := #Timers.UnloadTimer.Q;
	END_REGION
	
	//Set AutoMode off
	IF #R_TRIG_Stop.Q THEN
	    #Local.AutoMode := FALSE;
	END_IF;
	
	//Error trig
	IF #R_TRIG_CriticalError.Q THEN
	    IF NOT #PositioningAxis_Instance.Status.Done THEN
	        #Local.isMoved := TRUE;
	    END_IF;
	
	    "changeState"(newState := #S_ERROR,
	                  Data := #State);
	END_IF;
	
	REGION Change state
	    IF #State.inputFlag AND NOT #State.outputFlag THEN
	        #State.inputFlag := FALSE;
	    END_IF;
	    #State.outputFlag := FALSE;
	END_REGION
END_FUNCTION_BLOCK

